		//If valid destination found
		IF(_MPD.CV[CvIndex].DepositFuncNumber <> E_FunctionNumber.F_BEGIN_FUNCTION) THEN
			_MPD.CV[CvIndex].HighestPriority := TRUE;
			_MPD.CV[CvIndex].State := E_MPD_CvStates.E_CV_OCCUPIED;
			IF(_DebugPrint) THEN _M_DebugPrint(0,'Recover->E_CV_OCCUPIED'); END_IF
			_M_GetPickupDepositFunctions := TRUE;
		END_IF
	ELSE	    
		//Normal functionality, get prioritized data  	
		_MPD.CV[CvIndex].PickupFuncNumber 	:= rPrioFunctions.PickupFunctionNumber;
		_MPD.CV[CvIndex].DepositFuncNumber 	:= rPrioFunctions.DepositFunctionNumber;
		_MPD.CV[CvIndex].HighestPriority 	:= rPrioFunctions.HighestPriority;
		_M_GetPickupDepositFunctions := TRUE;
	END_IF
ELSE
	_MPD.CV[CvIndex].PickupFuncNumber 	:= E_FunctionNumber.F_BEGIN_FUNCTION; 
	_MPD.CV[CvIndex].DepositFuncNumber 	:= E_FunctionNumber.F_BEGIN_FUNCTION;
	_MPD.CV[CvIndex].HighestPriority 	:= FALSE;
END_IF
END_METHOD

METHOD PRIVATE _M_IsErrorActive : BOOL

_M_IsErrorActive :=ElementData.ErrorData.FunctionErrorPending OR ElementData.ErrorData.ErrorState = E_ErrorState.ERROR;
END_METHOD

//check if Pickup or Deposit function is in error during takover or handover or if element is stoped
METHOD PRIVATE _M_IsErrorActiveOnPD : BOOL
VAR_INPUT
END_VAR
VAR
	i:INT;
	myElementNumber		: E_ElementNumber;
	myFunctionNumbers	: ARRAY [1..4] OF E_FunctionNumber;
END_VAR

//only check if an transport is activated
IF(_MPD.CV[GVL_MPD.CV_A].State = E_MPD_CvStates.E_CV_PICKUP) THEN
	myFunctionNumbers[1] := _MPD.CV[GVL_MPD.CV_A].PickupFuncNumber;
END_IF
IF(_MPD.CV[GVL_MPD.CV_A].State = E_MPD_CvStates.E_CV_DEPOSIT) THEN
	myFunctionNumbers[2] := _MPD.CV[GVL_MPD.CV_A].DepositFuncNumber;	
END_IF
IF(_MPD.CV[GVL_MPD.CV_B].State = E_MPD_CvStates.E_CV_PICKUP) THEN
	myFunctionNumbers[3] := _MPD.CV[GVL_MPD.CV_B].PickupFuncNumber;
END_IF
IF(_MPD.CV[GVL_MPD.CV_B].State = E_MPD_CvStates.E_CV_DEPOSIT) THEN
	myFunctionNumbers[4] := _MPD.CV[GVL_MPD.CV_B].DepositFuncNumber;
END_IF

(**************************************************************************************************************
//check that the deposit element, function or zone is in error	
**************************************************************************************************************)
FOR i:=1 TO 4 DO	
	IF(__ISVALIDREF(FunctionRegistry[myFunctionNumbers[i]].rSettingsFunction)) THEN
		myElementNumber := FunctionRegistry[myFunctionNumbers[i]].rSettingsFunction.eElementLink;
		IF(__ISVALIDREF(ElementRegistry[myElementNumber].rElementData))THEN
			IF(	ElementRegistry[myElementNumber].rElementData.ErrorData.FunctionErrorPending OR
				ElementRegistry[myElementNumber].rElementData.ErrorData.ErrorState = E_ErrorState.ERROR OR
				ElementRegistry[myElementNumber].rElementData.OperationState.eState = E_PositionState.STOPPED) THEN
				_M_IsErrorActiveOnPD := TRUE; //an error occured during and active TU transport (handover or takeover)
				EXIT; // no need to loock further
			END_IF		
		END_IF		
	END_IF
END_FOR
END_METHOD

METHOD PRIVATE _M_MPD_CvStates : BOOL
VAR_INPUT
	CvIndex 	: INT;  // 1=A, 2=B
END_VAR

CASE _MPD.CV[CvIndex].State OF
	
	E_MPD_CvStates.E_CV_INIT:		
		_MPD.CV[CvIndex].PickupFuncNumber := _MPD.CV[CvIndex].DepositFuncNumber := E_FunctionNumber.F_BEGIN_FUNCTION;
		_MPD.CV[CvIndex].HighestPriority := FALSE;		
		_MPD.CV[CvIndex].State := E_MPD_CvStates.E_CV_IDLE;
		IF(_DebugPrint) THEN _M_DebugPrint(CvIndex,'Idle');END_IF
		
	
	// idle, cv waiting for job assignment.
	E_MPD_CvStates.E_CV_IDLE:		
		
		IF _EntryReqActive OR _EntryModeActive OR ElementData.OperationState.eMode <> E_PositionMode.AUTO_MODE OR ElementData.OperationState.eState <> E_PositionState.STARTED THEN
			;//Do Nothing
		ELSIF (_MPD.CV[CvIndex].PickupFuncNumber <> E_FunctionNumber.F_BEGIN_FUNCTION AND _MPD.CV[CvIndex].DepositFuncNumber <> E_FunctionNumber.F_BEGIN_FUNCTION) THEN
				_MPD.CV[CvIndex].State := E_MPD_CvStates.E_CV_JOBASSIGNED;		
		ELSE
			//Get prioritized pickup and deposit function
			_M_GetPickupDepositFunctions(CvIndex, FALSE);			
		END_IF
		
		
	//Shuttle Conveyor has a job assigned, wait for shuttle to get into correct position
	E_MPD_CvStates.E_CV_JOBASSIGNED:
		//check that pickup position still is valid
		IF(NOT  _M_GetPickupDepositFunctions(CvIndex,TRUE(*Verify*))) THEN
			_MPD.CV[CvIndex].State := E_MPD_CvStates.E_CV_INIT;
		ELSIF( _MPD.CV[CvIndex].PosPickupReached) THEN			
			//ElementRegistry[E_ElementNumber.E_11_002_0206_00_0].rElement.fbDebugMsg.M_SendInfoMsg(CONCAT(CONCAT('Shuttle: ', GVL_MPD.CV_IxNAME[CvIndex]),CONCAT('. Pickup adjacent function: ', F_GetFunctionName(_SC.CV[CvIndex].PickupFuncNumber,0))));			
			_MPD.CV[CvIndex].State := E_MPD_CvStates.E_CV_PICKUP;			
		END_IF
	
	//Wait for pickup to be complete. ie transfer TU from pickup function on to the shuttle conveyor
	E_MPD_CvStates.E_CV_PICKUP:
		//Set links for  pickup adjacent function, to point towards correct Shuttle conveyor (CV A or CV B)
		_M_SetLinks(CvIndex,TRUE,FALSE,FALSE,ElementData.ErrorData.ErrorDataSet[7]);		
		IF(NOT CtrlIn.HoldPosition AND _M_CheckTransportComplete(_MPD.CV[CvIndex].State, CvIndex)) THEN 
			_MPD.CV[CvIndex].State := E_MPD_CvStates.E_CV_OCCUPIED;
			IF(_DebugPrint) THEN _M_DebugPrint(CvIndex,'->E_CV_OCCUPIED');END_IF
		END_IF
	
	// pickup complete, and shuttle conveyor occupied, wait for deposit function is reached
	E_MPD_CvStates.E_CV_OCCUPIED:
		//incase of recovery from abnormal shutdown or Semi Auto Mode
		IF(NOT _MPD.RequestMove OR _MPD.State = E_MPD_States.E_SEMI_MODE) THEN
			;//Wait 
		ELSIF( _MPD.CV[CvIndex].PosDepositReached) THEN
			//restore Pickup adjacent function to default
			_M_SetLinks(CvIndex,TRUE,FALSE,TRUE,ElementData.ErrorData.ErrorDataSet[7]);		
			IF(_DebugPrint) THEN _M_DebugPrint(CvIndex,CONCAT('->E_CV_DEPOSIT to function: ', F_GetFunctionName(_MPD.CV[CvIndex].DepositFuncNumber,0))); END_IF				
			_MPD.CV[CvIndex].State := E_MPD_CvStates.E_CV_DEPOSIT;
		END_IF
	
	E_MPD_CvStates.E_CV_DEPOSIT:	
		//incase of recovery from abnormal shutdown or Semi Auto Mode
		IF(NOT _MPD.RequestMove OR _MPD.State = E_MPD_States.E_SEMI_MODE) THEN
			_MPD.CV[CvIndex].State := E_MPD_CvStates.E_CV_OCCUPIED;
			IF(_DebugPrint) THEN _M_DebugPrint(CvIndex,'->E_CV_OCCUPIED'); END_IF
		END_IF
		//Set links for the deposit adjacent function, to point towards correct Shuttle conveyor (CV A or CV B)
		_M_SetLinks(CvIndex,FALSE,TRUE,FALSE,ElementData.ErrorData.ErrorDataSet[7]);		
		IF(NOT CtrlIn.HoldPosition AND _M_CheckTransportComplete(_MPD.CV[CvIndex].State, CvIndex)) THEN
			//restore deposit adjacent function to default
			_M_SetLinks(CvIndex,FALSE,TRUE,TRUE,ElementData.ErrorData.ErrorDataSet[7]);
			IF(_DebugPrint) THEN _M_DebugPrint(CvIndex,'->E_CV_DONE'); END_IF
			_MPD.CV[CvIndex].State := E_MPD_CvStates.E_CV_DONE;
		END_IF
	
	E_MPD_CvStates.E_CV_DONE:		
		IF(_MPD.State = E_MPD_States.E_CYCLE_COMPLETE) THEN						
			_MPD.CV[CvIndex].State := E_MPD_CvStates.E_CV_INIT;
		END_IF
	
	ELSE
		F_SetError( ErrorType:= E_ErrorType.ERROR, 	ErrorParam:= '_M_ShuttleCvStates sequence error' , ErrorMsg:= E_ErrorConv.SOFTWARE_ERROR, ErrorData:= ElementData.ErrorData.ErrorDataSet[7]);
	
END_CASE
END_METHOD

METHOD PRIVATE _M_MPD_Init : BOOL
VAR
	EmptyShuttleConv 	: ST_MPD_CV;
	i,j 				: INT;
	InitSuccess 		: BOOL :=TRUE;
END_VAR

VAR_INST
	InitDelay : TON; // Startup delay for the function(s) connected to the element to initialize 
END_VAR
// Init function, performed once at init
_MPD.CV[GVL_MPD.CV_A] := EmptyShuttleConv;
_MPD.CV[GVL_MPD.CV_B] := EmptyShuttleConv;
_MPD.State := 0;

//_SC.ShuttleFuncNumber					:= ElementData ConfigFunction.eFunctionNumber;
_MPD.CV[GVL_MPD.CV_A].CvFuncNumber	:= ElementData.MemberList.FunctionList[1].eFunctionNumber;
_MPD.CV[GVL_MPD.CV_B].CvFuncNumber	:= ElementData.MemberList.FunctionList[2].eFunctionNumber;

_MPD.CV[GVL_MPD.CV_A].Enabled		:= _MPD.CV[GVL_MPD.CV_A].CvFuncNumber <> E_FunctionNumber.F_BEGIN_FUNCTION;
_MPD.CV[GVL_MPD.CV_B].Enabled		:= _MPD.CV[GVL_MPD.CV_B].CvFuncNumber <> E_FunctionNumber.F_BEGIN_FUNCTION;
// Check if there is a Pick Desposit
IF(MPD_Config.MPD_Type = E_MotionPD_Type.E_Unknown) THEN
	F_SetError(ErrorType:= E_ErrorType.ERROR, 
				ErrorParam:= 'Motion PD type not defined', 
				ErrorMsg:= E_ErrorConv.CONFIGURATION_ERROR, 
				ErrorData:= ElementData.ErrorData.ErrorDataSet[NUMBER_OF_ERROR_SETS]); 
	InitSuccess:=FALSE;
END_IF
// -Check correct assignment in. Element has at least has a shuttle function + minimum one additional function
InitDelay(IN:=TRUE,PT:=T#10S);
IF(_MPD.CV[GVL_MPD.CV_A].CvFuncNumber = E_FunctionNumber.F_BEGIN_FUNCTION AND _MPD.CV[GVL_MPD.CV_B].CvFuncNumber = E_FunctionNumber.F_BEGIN_FUNCTION) THEN
	IF(InitDelay.Q) THEN
		F_SetError(ErrorType:= E_ErrorType.ERROR, 
					ErrorParam:= 'Element has not assigned CvA to an function', 
					ErrorMsg:= E_ErrorConv.CONFIGURATION_ERROR, 
					ErrorData:= ElementData.ErrorData.ErrorDataSet[NUMBER_OF_ERROR_SETS]); 
		InitDelay(IN:=FALSE);
	END_IF
	InitSuccess:=FALSE;
	RETURN;
END_IF
// Check configuration
// -Check that not the same function is assigned more than once
FOR i := 1 TO GVL_MPD.MAXPDs - 1 BY 1 DO 
	FOR j := i + 1 TO GVL_MPD.MAXPDs BY 1 DO
		IF (MPD_Config.ConvCFG[i].eFunctionNumber = MPD_Config.ConvCFG[j].eFunctionNumber  AND MPD_Config.ConvCFG[i].eFunctionNumber<>E_FunctionNumber.F_BEGIN_FUNCTION) THEN
			F_SetError(ErrorType:= E_ErrorType.ERROR, 
				ErrorParam:= CONCAT('Doublets configured in Config.ConvCFG index: ', INT_TO_STRING(i)) , 
				ErrorMsg:= E_ErrorConv.CONFIGURATION_ERROR, 
				ErrorData:= ElementData.ErrorData.ErrorDataSet[NUMBER_OF_ERROR_SETS]); 
				InitSuccess := FALSE;
		END_IF
	END_FOR
END_FOR
// Check configuration
// -check at least one of the EnableConv parameters are set
FOR i := 1 TO GVL_MPD.MAXPDs - 1 BY 1 DO	
	IF (MPD_Config.ConvCFG[i].eFunctionNumber <> E_FunctionNumber.F_BEGIN_FUNCTION AND
		(MPD_Config.ConvCFG[i].EnableConv[1]=FALSE AND  MPD_Config.ConvCFG[i].EnableConv[2]=FALSE)) THEN
			F_SetError(ErrorType:= E_ErrorType.ERROR, 
				ErrorParam:= CONCAT('Both EnableConv[x] in Config.ConvCFG index: ', INT_TO_STRING(i)) , 
				ErrorMsg:= E_ErrorConv.CONFIGURATION_ERROR, 
				ErrorData:= ElementData.ErrorData.ErrorDataSet[NUMBER_OF_ERROR_SETS]); 
				InitSuccess := FALSE;
	END_IF	
END_FOR	
// Check configuration
// -check that position is set within the valid range
FOR i := 1 TO GVL_MPD.MAXPDs - 1 BY 1 DO 
	FOR j:=GVL_MPD.CV_A TO GVL_MPD.CV_B DO
		IF (MPD_Config.ConvCFG[i].eFunctionNumber <> E_FunctionNumber.F_BEGIN_FUNCTION AND
			(MPD_Config.ConvCFG[i].EnableConv[j] AND (MPD_Config.ConvCFG[i].PositionConv < MPD_Config.DriveCFG.MinimumPosition OR MPD_Config.ConvCFG[i].PositionConv>MPD_Config.DriveCFG.MaximumPosition))) THEN
				F_SetError(ErrorType:= E_ErrorType.ERROR, 
					ErrorParam:= CONCAT('PositionConv in Config.ConvCFG index: ', INT_TO_STRING(i)), 
					ErrorMsg:= E_ErrorConv.CONFIGURATION_ERROR, 
					ErrorData:= ElementData.ErrorData.ErrorDataSet[NUMBER_OF_ERROR_SETS]); 
					InitSuccess := FALSE;
		END_IF
	END_FOR	
END_FOR
// Check the for invalid homing function should not be F_BegainFunction or set an error
IF MPD_Config.EncoderHoming.HomingFunctionNumber = E_FunctionNumber.F_BEGIN_FUNCTION AND MPD_Config.EncoderHoming.HomingEnable THEN
	F_SetError(ErrorType:= E_ErrorType.ERROR, 
					ErrorParam:= 'Invalid Homing Function number', 
					ErrorMsg:= E_ErrorConv.CONFIGURATION_ERROR, 
					ErrorData:= ElementData.ErrorData.ErrorDataSet[NUMBER_OF_ERROR_SETS]); 
					InitSuccess := FALSE;
END_IF	
// Check configuration
// Check pickup position offset
FOR i := 1 TO GVL_MPD.MAXPDs - 1 BY 1 DO 
	FOR j:=GVL_MPD.CV_A TO GVL_MPD.CV_B DO
		IF (MPD_Config.ConvCFG[i].eFunctionNumber <> E_FunctionNumber.F_BEGIN_FUNCTION AND MPD_Config.ConvCFG[i].EnableConv[j]) THEN
			
			IF(MPD_Config.MPD_Type = E_MotionPD_Type.E_ShuttleCar) THEN
				//PickupPositionOffset must be zero for shuttle cars
				IF(MPD_Config.MPD_Type = E_MotionPD_Type.E_ShuttleCar AND MPD_Config.ConvCFG[i].PickupPositionOffset<>0) THEN
					 F_SetError(ErrorType:= E_ErrorType.ERROR, 
						ErrorParam:= CONCAT('PickupPositionOffset<>0 . Config.ConvCFG index: ', INT_TO_STRING(i)), 
						ErrorMsg:= E_ErrorConv.CONFIGURATION_ERROR, 
						ErrorData:= ElementData.ErrorData.ErrorDataSet[NUMBER_OF_ERROR_SETS]); 
						InitSuccess := FALSE;
				END_IF
				//DepsitPositionOffset must be zero for shuttle cars
				 IF(MPD_Config.MPD_Type = E_MotionPD_Type.E_ShuttleCar AND MPD_Config.ConvCFG[i].DepsitPositionOffset<>0) THEN
					 F_SetError(ErrorType:= E_ErrorType.ERROR, 
						ErrorParam:= CONCAT('DepsitPositionOffset<>0 . Config.ConvCFG index: ', INT_TO_STRING(i)), 
						ErrorMsg:= E_ErrorConv.CONFIGURATION_ERROR, 
						ErrorData:= ElementData.ErrorData.ErrorDataSet[NUMBER_OF_ERROR_SETS]); 
						InitSuccess := FALSE;
				END_IF
			END_IF
			
			IF(MPD_Config.MPD_Type = E_MotionPD_Type.E_VerticalCv) THEN
				//PickupPositionOffset must be sane. ie between -200 and + 200
				IF(MPD_Config.ConvCFG[i].PickupPositionOffset > 200 AND MPD_Config.ConvCFG[i].PickupPositionOffset <-200) THEN
					F_SetError(ErrorType:= E_ErrorType.ERROR, 
						ErrorParam:= CONCAT('PickupPositionOffset +-200 in Config.ConvCFG index: ', INT_TO_STRING(i)), 
						ErrorMsg:= E_ErrorConv.CONFIGURATION_ERROR, 
						ErrorData:= ElementData.ErrorData.ErrorDataSet[NUMBER_OF_ERROR_SETS]); 
						InitSuccess := FALSE;
				END_IF
			END_IF
		END_IF
	END_FOR	
END_FOR
// Check CVCC, must be 0 for VC type
IF(MPD_Config.MPD_Type = E_MotionPD_Type.E_VerticalCv AND MPD_Config.CvCC <> 0) THEN
	F_SetError(ErrorType:= E_ErrorType.ERROR, 
				ErrorParam:= 'MPD_Config.CvCC must be set to 0', 
				ErrorMsg:= E_ErrorConv.CONFIGURATION_ERROR, 
				ErrorData:= ElementData.ErrorData.ErrorDataSet[NUMBER_OF_ERROR_SETS]); 
	InitSuccess:=FALSE;
END_IF

_M_MPD_Init := InitSuccess;
END_METHOD

METHOD PROTECTED _M_MPD_Mover : BOOL
VAR_INPUT
END_VAR
VAR
	i					: INT;
	DesiredPos			: DINT;	
	MoviDriveManual		: ST_MoviDriveManual;
END_VAR

VAR_INST
	CVInPosTimeout		: TON;//if position is not correct stop, set an error	
	ScMoveTimeout		: TON := (PT:=T#30S);	//Shuttle Car Move Timeout
	EntryReqState		: INT;
END_VAR

CASE EntryReqState OF
	0:	//Trig an entry request..
		IF(CtrlIn.RequestEntry) THEN 
			_EntryReqActive :=TRUE;
			EntryReqState := EntryReqState+1;
		END_IF
	1: // wait for position is reached
		IF(_MPD.EntryPosReached) THEN
			_EntryModeActive :=TRUE;
			_EntryReqActive :=FALSE;
			EntryReqState := EntryReqState+1;
		END_IF
	2: // Entry pos is reched, wait for operator to turn off key
		IF(NOT CtrlIn.RequestEntry) THEN
			_EntryModeActive :=FALSE;
			EntryReqState := EntryReqState+1;
		END_IF
	ELSE
		EntryReqState := 0;	
END_CASE


// Call Shuttle car mover...
// Manual Control
IF(_MPD.State = E_MPD_States.E_SEMI_MODE AND CtrlIn.SemiDriveCtrl.SemiManualMode) THEN 
	//Semi manual control
	MoviDriveManual.DriveFwd := CtrlIn.SemiDriveCtrl.SemiControlFWD;
	MoviDriveManual.DriveRev := CtrlIn.SemiDriveCtrl.SemiControlREV;
	MoviDriveManual.EmergencyDrive := FALSE;
ELSE
	//Normal Manual control
	MoviDriveManual.DriveFwd := HW_Inputs.ManualControl.DriveFwd;
	MoviDriveManual.DriveRev := HW_Inputs.ManualControl.DriveRev;
	MoviDriveManual.EmergencyDrive := HW_Inputs.ManualControl.EmergencyDrive;
END_IF



IF( NOT ProBoxSystem.EMULATION_ENABLED) THEN	
		
	//Request to move Normal operation
	IF _MPD.RequestMove AND NOT _EntryModeActive THEN 
		fbMPDMover.M_MoveAbsolute(
			mPosition		:= _MPD.RequestPosValue, 
			mVelocity		:= MPD_Config.DriveCFG.DriveParameter[_MPD.DriveParameterIndex].Velocity, 
			mAcceleration	:= MPD_Config.DriveCFG.DriveParameter[_MPD.DriveParameterIndex].Acceleration, 
			mDeceleration	:= MPD_Config.DriveCFG.DriveParameter[_MPD.DriveParameterIndex].Deceleration, 
			mJerk			:= MPD_Config.DriveCFG.DriveParameter[_MPD.DriveParameterIndex].Jerk,
			ErrorData 		:= ElementData.ErrorData.ErrorDataSet[5]);
	
	//Request move to entry
	ELSIF _EntryReqActive AND NOT _MPD.RequestMove AND _MPD.State = E_MPD_States.E_IDLE THEN 
		fbMPDMover.M_MoveAbsolute(
			mPosition		:= CtrlIn.RequestEntryPos, //EntryPosition, 
			mVelocity		:= MPD_Config.DriveCFG.DriveParameter[_MPD.DriveParameterIndex].Velocity, 
			mAcceleration	:= MPD_Config.DriveCFG.DriveParameter[_MPD.DriveParameterIndex].Acceleration, 
			mDeceleration	:= MPD_Config.DriveCFG.DriveParameter[_MPD.DriveParameterIndex].Deceleration, 
			mJerk			:= MPD_Config.DriveCFG.DriveParameter[_MPD.DriveParameterIndex].Jerk,
			ErrorData 		:= ElementData.ErrorData.ErrorDataSet[5]);
	END_IF
	
	fbMPDMover(
		ErrorPending			:= _M_IsErrorActive(), 
		ElementOperationState	:= ElementData.OperationState,
		DisableEnableDrive 		:= (NOT _MPD.RequestMove AND NOT _EntryReqActive) OR _M_IsErrorActiveOnPD(), 
		DriveCFG				:= MPD_Config.DriveCFG,
		ManualControl			:= MoviDriveManual,		  
		DriveInputs				:= HW_Inputs.DriveInputs,		
		EmgStopAxisTrig 		:= EmergencyStop,
		Done 					=> _MPD.Locked, 
		Aborted 				=> _MPD.MotionAborted,
		ErrorData 				:= ElementData.ErrorData.ErrorDataSet[5]);
	
	
	
	_MPD.ActualPosValue := LREAL_TO_DINT( fbMPDMover.ActPos);
END_IF	
	

//-----------------------------------------------------------------------------
// Set interface variables used in ShuttleState and ShuttleCVStates
//-----------------------------------------------------------------------------
FOR i:=GVL_MPD.CV_A TO GVL_MPD.CV_B DO
			
	//Pickup position reached?
	DesiredPos := M_GetDesiredPosition(_MPD.CV[i].PickupFuncNumber, i, TRUE,FALSE);
	_MPD.CV[i].PosPickupReached := M_CheckDesiredPosition(DesiredPos) AND _MPD.Locked AND _MPD.RequestMove AND _MPD.CV[i].PickupFuncNumber > E_FunctionNumber.F_BEGIN_FUNCTION;
	
	//Deposit position reached?
	DesiredPos := M_GetDesiredPosition(_MPD.CV[i].DepositFuncNumber, i, FALSE, TRUE);	
	_MPD.CV[i].PosDepositReached := M_CheckDesiredPosition(DesiredPos) AND _MPD.Locked AND _MPD.RequestMove AND _MPD.CV[i].DepositFuncNumber > E_FunctionNumber.F_BEGIN_FUNCTION;
END_FOR

	//Idle Position reached?
	_MPD.IdlePosReached := M_CheckDesiredPosition(MPD_Config.IdlePosition) AND _MPD.Locked AND MPD_Config.EnableIdlePosition;

	//Entry Position reached?
	_MPD.EntryPosReached := M_CheckDesiredPosition(CtrlIn.RequestEntryPos) AND _MPD.Locked;

//-----------------------------------------------------------------------------	
// Error handling: Check car movement is performed within acceptable time 
//-----------------------------------------------------------------------------	
	
//Check shuttle Car movement Timeout
ScMoveTimeout(IN:=_MPD.RequestMove AND NOT _MPD.Locked AND (ElementData.OperationState.eState = E_PositionState.STARTED OR ElementData.OperationState.eState = E_PositionState.STOPPING), 
				PT:= MPD_Config.TimeOutMove);
IF(ScMoveTimeout.Q) THEN
	F_SetError( ErrorType:= E_ErrorType.ERROR, 	ErrorParam:= 'Movement Timeout' , (* Could not get to the destination with in expected time*) 
				ErrorMsg:= E_ErrorConv.TIMEOUT, ErrorData:= ElementData.ErrorData.ErrorDataSet[4]);
	ScMoveTimeout(IN:=FALSE);
END_IF


//-----------------------------------------------------------------------------	
// Error handling: Timeout during takeover or handover. Note: the Shuttle car servo shall stop immediately
// If element is not in error and not adjacent function, then it is somthiing else that makes the transport not possible to finalize (could be that the deposit function is disabled..)
//-----------------------------------------------------------------------------
CVInPosTimeout(	IN:= NOT _M_IsErrorActive() AND NOT _M_IsErrorActiveOnPD() AND _MPD.RequestMove AND ( _MPD.State = E_MPD_States.E_PICKINGUP OR _MPD.State = E_MPD_States.E_DEPOSITING),
				PT:= MPD_Config.TimeOutMove); 
IF(CVInPosTimeout.Q) THEN		 
	F_SetError(E_ErrorType.ERROR,'Timeout during Pickup or deposit',E_ErrorConv.TIMEOUT,ElementData.ErrorData.ErrorDataSet[4]);
END_IF 

	
//-----------------------------------------------------------------------------
//Emulation shuttle car posioning
//-----------------------------------------------------------------------------
END_METHOD

METHOD PRIVATE _M_MPD_States : BOOL
VAR_INPUT
END_VAR


VAR	
	i		: INT;
	OtherCv	: ARRAY[1..2] OF INT := [GVL_MPD.CV_B,GVL_MPD.CV_A];	
END_VAR

VAR_INST
	EnterIdlePosTmr		: TON := (PT:= T#2S); //delay before entering Idle position	
END_VAR
EnterIdlePosTmr();


CASE _MPD.State OF
	
	//---------------------------------------------------------------------------------------------------
	E_MPD_States.E_INIT:
		_MPD.RequestMove := FALSE;
		_MPD.State:=E_MPD_States.E_IDLE;
		
	
		
	//---------------------------------------------------------------------------------------------------
	// Waiting for job to do	
	E_MPD_States.E_IDLE: 
		EnterIdlePosTmr.IN:=FALSE;
		_M_AutoAdjustVCHeight(FALSE,FALSE,TRUE (*Reset*), FALSE);
				
		//Check if we can proceed...
		IF(ElementData.OperationState.eState <> E_PositionState.STARTED OR ElementData.OperationState.eMode <> E_PositionMode.AUTO_MODE OR
		   _EntryReqActive OR _EntryModeActive)  THEN
			//do nothing, but wait
 			_MPD.RequestMove	:= FALSE;	
		
		//Semi automatic or semi manual mode
		ELSIF(CtrlIn.SemiDriveCtrl.SemiAutoMode OR CtrlIn.SemiDriveCtrl.SemiManualMode) THEN			
			_MPD.State := E_MPD_States.E_SEMI_MODE;			
			IF(_DebugPrint) THEN _M_DebugPrint(0,CONCAT('->E_SEMI_MODE : ', TO_STRING(_MPD.RequestPosValue))); END_IF
	
		//Normal operation, picking up
		ELSIF( _MPD.CV[GVL_MPD.CV_A].State = E_MPD_CvStates.E_CV_PICKUP OR _MPD.CV[GVL_MPD.CV_B].State = E_MPD_CvStates.E_CV_PICKUP) THEN 
			_MPD.State := E_MPD_States.E_PICKINGUP;
			
		//Normal operation, Depositing
		ELSIF( _MPD.CV[GVL_MPD.CV_A].State = E_MPD_CvStates.E_CV_DEPOSIT OR _MPD.CV[GVL_MPD.CV_B].State = E_MPD_CvStates.E_CV_DEPOSIT) THEN 
			_MPD.State := E_MPD_States.E_DEPOSITING;
			
		//Normal operation, check if an job is assigned to CV A or CV B
		ELSIF( _MPD.CV[GVL_MPD.CV_A].State = E_MPD_CvStates.E_CV_JOBASSIGNED OR _MPD.CV[GVL_MPD.CV_B].State = E_MPD_CvStates.E_CV_JOBASSIGNED) THEN		
			// Element has no error pending and wheres a job to do	
			_MPD.State := E_MPD_States.E_START_PICKUP;						
		
		//check if CV A or CV B is occupied
		ELSIF( _MPD.CV[GVL_MPD.CV_A].State = E_MPD_CvStates.E_CV_OCCUPIED OR _MPD.CV[GVL_MPD.CV_B].State = E_MPD_CvStates.E_CV_OCCUPIED) THEN	 
			_MPD.State := E_MPD_States.E_START_DEPOSIT;		
			
		//If no active jobs move to idle position	
		ELSIF (MPD_Config.EnableIdlePosition) THEN
			EnterIdlePosTmr.IN := NOT _MPD.IdlePosReached AND NOT _EntryReqActive AND NOT _M_IsErrorActive();
			IF(EnterIdlePosTmr.Q) THEN			
					// Set desired Shuttle car position
					_MPD.RequestPosValue := MPD_Config.IdlePosition;
					// Release shuttle car brake
					_MPD.RequestMove := TRUE;
			ELSE
				_MPD.RequestMove := FALSE;
			END_IF
		END_IF
	
	
	
		//---------------------------------------------------------------------------------------------------
		// Semi automatic mode	
		E_MPD_States.E_SEMI_MODE:
			IF ((NOT CtrlIn.SemiDriveCtrl.SemiAutoMode AND NOT CtrlIn.SemiDriveCtrl.SemiManualMode)OR
				(ElementData.OperationState.eMode <> E_PositionMode.AUTO_MODE)) THEN
				_MPD.RequestMove := FALSE;
				_MPD.State := E_MPD_States.E_IDLE;
				IF(_DebugPrint) THEN _M_DebugPrint(0,CONCAT('->E_IDLE : ', TO_STRING(_MPD.RequestPosValue))); END_IF		
			END_IF		
		
		
		
		
	//---------------------------------------------------------------------------------------------------
	// Decide prioirty for A and B	
	E_MPD_States.E_START_PICKUP:
				
		FOR i:=GVL_MPD.CV_A TO GVL_MPD.CV_B DO			
			IF( _M_IsErrorActive()=FALSE ) THEN  //element has no error pending
				IF(_MPD.CV[i].State = E_MPD_CvStates.E_CV_JOBASSIGNED AND (_MPD.CV[i].HighestPriority  OR _MPD.CV[OtherCv[i]].State = E_MPD_CvStates.E_CV_OCCUPIED))THEN
					// Set desired Shuttle car position
					_MPD.RequestPosValue := M_GetDesiredPosition(_MPD.CV[i].PickupFuncNumber, i, TRUE,FALSE);
					// Release shuttle car brake
					_MPD.RequestMove := TRUE;
					//move to next state
					_MPD.State := E_MPD_States.E_MOVE_TO_PICKUP;					
					IF(_DebugPrint) THEN _M_DebugPrint(0,CONCAT('->E_MOVE_TO_PICKUP : ', TO_STRING(_MPD.RequestPosValue))); END_IF
					EXIT;					
				END_IF	
			END_IF				
		END_FOR
		

	
	//---------------------------------------------------------------------------------------------------	
	E_MPD_States.E_MOVE_TO_PICKUP:
		
		IF(_MPD.CV[GVL_MPD.CV_A].State <> E_MPD_CvStates.E_CV_JOBASSIGNED AND _MPD.CV[GVL_MPD.CV_B].State <> E_MPD_CvStates.E_CV_JOBASSIGNED) THEN
			_MPD.State:=E_MPD_States.E_IDLE; //start over, Shuttle CV states may not be fulfiled anymore.  
		ELSE			
			//Check if shuttle car is in position
			FOR i:=GVL_MPD.CV_A TO GVL_MPD.CV_B DO
				IF(_MPD.CV[i].PosPickupReached ) THEN				
					//position reached				
					_MPD.State := E_MPD_States.E_PICKUP_POSITION_REACHED;				
					IF(_DebugPrint) THEN _M_DebugPrint(0,'->E_PICKUP_POSITION_REACHED'); END_IF	
					EXIT;			
				END_IF								
			END_FOR
		END_IF
			
		
		
	//---------------------------------------------------------------------------------------------------	
	E_MPD_States.E_PICKUP_POSITION_REACHED:
		//At this point only check that MPD locked the position, as the acutal position may change if AutoAdjustVCHeight is used.
		IF(_MPD.Locked AND NOT _MPD.MotionAborted) THEN
			_MPD.State := E_MPD_States.E_PICKINGUP;
		END_IF

	//---------------------------------------------------------------------------------------------------		
	E_MPD_States.E_PICKINGUP:
	
		//Adjust VC height
		_MPD.RequestPosValue := _MPD.RequestPosValue + _M_AutoAdjustVCHeight(TRUE,FALSE,FALSE,FALSE);
		//wait for pickup is complete
		//there can be a situation where we have a parallell transport of CvA and CvB, so wait till conveyors finishing transport
		IF (_MPD.CV[GVL_MPD.CV_A].State <> E_MPD_CvStates.E_CV_PICKUP AND _MPD.CV[GVL_MPD.CV_B].State <> E_MPD_CvStates.E_CV_PICKUP) THEN						
			_MPD.State:=E_MPD_States.E_IDLE; //start over, and see the other shuttle CV (CV_A or CV_B) should be picked up						
			IF(_DebugPrint) THEN _M_DebugPrint(0,'E_PICKINGUP->E_IDLE'); END_IF						
		END_IF
		
		//in case motion was aborted/interupted. it may be so that SC/VC position is changed, check position is maintained. 
		IF(_MPD.MotionAborted) THEN
			_MPD.State:=E_MPD_States.E_PICKUP_POSITION_REACHED;
			IF(_DebugPrint) THEN _M_DebugPrint(0,'E_PICKINGUP->E_PICKUP_POSITION_REACHED'); END_IF
		END_IF
		
	//---------------------------------------------------------------------------------------------------		
	E_MPD_States.E_START_DEPOSIT: 
			
		FOR i:=GVL_MPD.CV_A TO GVL_MPD.CV_B DO
			IF(_M_IsErrorActive()=FALSE AND _MPD.CV[i].State = E_MPD_CvStates.E_CV_OCCUPIED AND (_MPD.CV[i].HighestPriority OR _MPD.CV[OtherCv[i]].State = E_MPD_CvStates.E_CV_DONE))THEN				
				// reqest shuttle car position
				_MPD.RequestPosValue := M_GetDesiredPosition(_MPD.CV[i].DepositFuncNumber, i, FALSE,TRUE);
				// Release shuttle car brake
				_MPD.RequestMove := TRUE;
				_MPD.State := E_MPD_States.E_MOVE_TO_DEPOSIT;
				IF(_DebugPrint) THEN _M_DebugPrint(0,CONCAT('E_START_DEPOSIT->E_MOVE_TO_DEPOSIT : ',  TO_STRING(_MPD.RequestPosValue))); END_IF
				EXIT;
			END_IF				
		END_FOR
	
	
	//---------------------------------------------------------------------------------------------------
	//Check if shuttle car is in position for depositing		
	E_MPD_States.E_MOVE_TO_DEPOSIT:
		//Check if shuttle car is in position
		FOR i:=GVL_MPD.CV_A TO GVL_MPD.CV_B DO
			IF(_MPD.CV[i].PosDepositReached AND _MPD.CV[i].State = E_MPD_CvStates.E_CV_DEPOSIT) THEN //if deposit position is reached, and CV_A or CV_B has reacted				
				//position reached				
				_MPD.State := E_MPD_States.E_DEPOSIT_POSITION_REACHED;
				IF(_DebugPrint) THEN _M_DebugPrint(0,CONCAT('E_MOVE_TO_DEPOSIT->E_DEPOSIT_POSITION_REACHED: ', GVL_MPD.CV_IxNAME[i])); END_IF
				EXIT; //break for loop				
			END_IF			
		END_FOR
	
			
	//---------------------------------------------------------------------------------------------------		
	E_MPD_States.E_DEPOSIT_POSITION_REACHED:
	//At this point only check that MPD locked the position, as the acutal position may change if AutoAdjustVCHeight is used.
		IF(_MPD.Locked AND NOT _MPD.MotionAborted) THEN
			_MPD.State:=E_MPD_States.E_DEPOSITING;	
		END_IF
	
	//---------------------------------------------------------------------------------------------------	
	E_MPD_States.E_DEPOSITING:
		//incase of recovery from abnormal shutdown or Semi Auto Mode	
		IF(NOT _MPD.RequestMove) THEN
			_MPD.State := E_MPD_States.E_START_DEPOSIT;
		END_IF
	
		//Adjust VC height
		_MPD.RequestPosValue := _MPD.RequestPosValue + _M_AutoAdjustVCHeight(FALSE,TRUE,FALSE,FALSE);
		
		//wait for depositing is complete		
		FOR i:=GVL_MPD.CV_A TO GVL_MPD.CV_B DO
			IF ((_MPD.CV[i].State = E_MPD_CvStates.E_CV_PICKUP OR _MPD.CV[OtherCv[i]].State = E_MPD_CvStates.E_CV_PICKUP) OR 
				(_MPD.CV[i].State = E_MPD_CvStates.E_CV_DEPOSIT OR _MPD.CV[OtherCv[i]].State = E_MPD_CvStates.E_CV_DEPOSIT))THEN
				// in the case we do an pickup in parallell with deposit (shuttle with 2 conveyors)
				;// do nothing but wait.							
			ElSIF (_MPD.CV[i].State = E_MPD_CvStates.E_CV_DONE AND _MPD.CV[OtherCv[i]].State = E_MPD_CvStates.E_CV_OCCUPIED) THEN
				// Go back and set the next deposit position for the shuttle car
				_MPD.State:=E_MPD_States.E_START_DEPOSIT;  	
				IF(_DebugPrint) THEN _M_DebugPrint(0,'E_DEPOSITING->E_START_DEPOSIT'); END_IF 	
			ELSIF( (_MPD.CV[i].State = E_MPD_CvStates.E_CV_DONE AND _MPD.CV[otherCv[i]].State <= E_MPD_CvStates.E_CV_IDLE) OR
				   (_MPD.CV[i].State = E_MPD_CvStates.E_CV_DONE AND _MPD.CV[otherCv[i]].State = E_MPD_CvStates.E_CV_DONE)) THEN	
					//proceed to next step			
					_MPD.State:=E_MPD_States.E_CYCLE_COMPLETE;
					IF(_DebugPrint) THEN _M_DebugPrint(0,'E_DEPOSITING->E_CYCLE_COMPLETE'); END_IF
			END_IF
		END_FOR
		
		//in case motion was aborted/interupted. it may be so that SC/VC position is changed, check position is maintained. 
		IF(_MPD.MotionAborted) THEN
			_MPD.State:=E_MPD_States.E_DEPOSIT_POSITION_REACHED;
		END_IF
		
		
	//---------------------------------------------------------------------------------------------------
	E_MPD_States.E_CYCLE_COMPLETE:
				
		_MPD.State:=E_MPD_States.E_INIT;
		
	ELSE
		F_SetError( ErrorType:= E_ErrorType.ERROR, 	ErrorParam:= '_M_ShuttleStates sequence error' , ErrorMsg:= E_ErrorConv.SOFTWARE_ERROR, ErrorData:= ElementData.ErrorData.ErrorDataSet[7]);
	
END_CASE
END_METHOD

METHOD PROTECTED _M_SemiDriveControl : BOOL
VAR_INPUT
END_VAR

IF(_MPD.State <> E_MPD_States.E_SEMI_MODE) THEN
	MemSet(ADR(fbMPDMover.SemiDriveControl),0, SIZEOF(fbMPDMover.SemiDriveControl));
ELSE
	fbMPDMover.SemiDriveControl.SemiAutoMode			:= CtrlIn.SemiDriveCtrl.SemiAutoMode AND NOT CtrlIn.SemiDriveCtrl.SemiManualMode;
	fbMPDMover.SemiDriveControl.SemiManualMode 			:= CtrlIn.SemiDriveCtrl.SemiManualMode AND NOT CtrlIn.SemiDriveCtrl.SemiAutoMode;
	fbMPDMover.SemiDriveControl.SemiTrigMoveAbs		 	:= CtrlIn.SemiDriveCtrl.SemiAutoEnableDrive;
	fbMPDMover.SemiDriveControl.SemiAutoHalt 			:= CtrlIn.SemiDriveCtrl.SemiAutoHalt;	
	//set request move
	IF(fbMPDMover.SemiDriveControl.SemiAutoMode) THEN
		//Semi auto mode
		_MPD.RequestMove := CtrlIn.SemiDriveCtrl.SemiAutoEnableDrive;
		_MPD.RequestPosValue := CtrlIn.SemiDriveCtrl.SemiAutoPositionToGo;					
	ELSE
		//Semi Man mode
		_MPD.RequestMove := FALSE;
	END_IF
	
	//Reset input variables in case user did'nt...
	CtrlIn.SemiDriveCtrl.SemiAutoHalt 					:= FALSE;
	IF(fbMPDMover.PositioningState = E_PositioningState.POSITIONING_ABSOLUTE) THEN	
		CtrlIn.SemiDriveCtrl.SemiAutoEnableDrive			:= FALSE;	
	END_IF
END_IF
END_METHOD

// Replace the deposit or pickup position adjacent functionnumber to point toward CVA or CVB
METHOD PRIVATE _M_SetAdjacentFunction : BOOL
VAR_INPUT
	ScCvFunction		: E_FunctionNumber; //the shuttle car conveyor function
	AdjacentFunction	: E_FunctionNumber; //the pickup or deposit function to change
	SearchFunctions		: ARRAY[1..3] OF E_FunctionNumber;
	RestoreToDefault	: BOOL;
END_VAR

VAR
	rFuncSettings  	: REFERENCE TO ST_CFG_Function;		//the pickup or deposit function where to replace the adjacent side
	rConfigSettings	: REFERENCE TO ST_CFG_Function;
	i:INT;
END_VAR

//

rFuncSettings REF= FunctionRegistry[AdjacentFunction].rSettingsFunction;
rConfigSettings REF= FunctionRegistry[AdjacentFunction].rFunction.ConfigFunction; 

//Replace the adjacent side of the deposit function to point towards the Shuttle conveyor A
IF(__ISVALIDREF(rFuncSettings) AND __ISVALIDREF(rConfigSettings)) THEN
	IF(NOT RestoreToDefault) THEN
		FOR i:= 1 TO 4 DO
			IF(	rFuncSettings.eAdjacentFunctionNumberSide[i] <> E_FunctionNumber.F_BEGIN_FUNCTION AND
				(rFuncSettings.eAdjacentFunctionNumberSide[i] = SearchFunctions[1] OR
				 rFuncSettings.eAdjacentFunctionNumberSide[i] = SearchFunctions[2] OR
				 rFuncSettings.eAdjacentFunctionNumberSide[i] = SearchFunctions[3] )) THEN
				 
					rFuncSettings.eAdjacentFunctionNumberSide[i] := ScCvFunction;
					_M_SetAdjacentFunction :=TRUE;
					//EXIT;
			END_IF			
		END_FOR
	// restore to default
	ELSE 
		rFuncSettings.eAdjacentFunctionNumberSide := rConfigSettings.eAdjacentFunctionNumberSide;				
	END_IF	
	
END_IF
END_METHOD

// Setup links, adjacent sides on shuttle car towards the pickup and deposition funciton
METHOD PRIVATE _M_SetLinks : BOOL
VAR_INPUT
	//CvAFuncNumb		: E_FunctionNumber;
	SC_CV_Index 		: INT; // 1 = A, 2 = B  
	SetPickupLinks		: BOOL; 
	SetDepositLinks		: BOOL; 
	RestorToDefault		: BOOL;
END_VAR
VAR_IN_OUT
	ErrorData 				: ST_ErrorDataSet; // Error data
END_VAR
VAR
	ReplaceFunctions	: ARRAY[1..3] OF E_FunctionNumber;	
END_VAR
	ReplaceFunctions[1] := _MPD.CV[GVL_MPD.CV_A].CvFuncNumber;	//the Shuttle Car Conveyor A functionNumber
	ReplaceFunctions[2] := _MPD.CV[GVL_MPD.CV_B].CvFuncNumber;	//the Shuttle Car Conveyor B functionNumber
	ReplaceFunctions[3] := E_FunctionNumber.F_BEGIN_FUNCTION;	//Spare, to remove?
	
	
	//Sanity check
	IF( NOT __ISVALIDREF(FunctionRegistry[_MPD.CV[SC_CV_Index].CvFuncNumber].rSettingsFunction)) THEN
		F_SetError(	ErrorType := E_ErrorType.ERROR,	ErrorParam := 'Setup Pickup transport link',ErrorMsg := E_ErrorConv.INCORRECT_POSITION, ErrorData := ErrorData);
		_M_SetLinks:= FALSE;
		RETURN;
	END_IF
		
	IF(NOT RestorToDefault AND SetPickupLinks) THEN		
		//Setup SettingsFunctions parameters for shuttle car conveyor		
		FunctionRegistry[_MPD.CV[SC_CV_Index].CvFuncNumber].rSettingsFunction.ePrevFunctionNumber := _MPD.CV[SC_CV_Index].PickupFuncNumber;
		FunctionRegistry[_MPD.CV[SC_CV_Index].CvFuncNumber].rSettingsFunction.eNextFunctionNumber := E_FunctionNumber.F_BEGIN_FUNCTION;
		
		//Set adjacent sides on shuttle conveyor	
		IF( M_GetConveyorDirection(_MPD.CV[SC_CV_Index].PickupFuncNumber) = E_PickupDepositSide.LeftSide) THEN
			//Pickup on left side -> drive Forward 
			FunctionRegistry[_MPD.CV[SC_CV_Index].CvFuncNumber].rSettingsFunction.eAdjacentFunctionNumberSide[1] := _MPD.CV[SC_CV_Index].PickupFuncNumber;
			FunctionRegistry[_MPD.CV[SC_CV_Index].CvFuncNumber].rSettingsFunction.eAdjacentFunctionNumberSide[2] := E_FunctionNumber.F_BEGIN_FUNCTION;	
		ELSE                 
			//Pickup on right side -> drive Reverse
			FunctionRegistry[_MPD.CV[SC_CV_Index].CvFuncNumber].rSettingsFunction.eAdjacentFunctionNumberSide[1] := E_FunctionNumber.F_BEGIN_FUNCTION;
			FunctionRegistry[_MPD.CV[SC_CV_Index].CvFuncNumber].rSettingsFunction.eAdjacentFunctionNumberSide[2] := _MPD.CV[SC_CV_Index].PickupFuncNumber;					
		END_IF		
	END_IF
	
	IF(NOT RestorToDefault AND SetDepositLinks) THEN
		//Setup SettingsFunctions parameters for shuttle car conveyor
		FunctionRegistry[_MPD.CV[SC_CV_Index].CvFuncNumber].rSettingsFunction.ePrevFunctionNumber := E_FunctionNumber.F_BEGIN_FUNCTION;		
		FunctionRegistry[_MPD.CV[SC_CV_Index].CvFuncNumber].rSettingsFunction.eNextFunctionNumber := _MPD.CV[SC_CV_Index].DepositFuncNumber;
		//Set adjacent sides on shuttle conveyor
		IF( M_GetConveyorDirection(_MPD.CV[SC_CV_Index].DepositFuncNumber) = E_PickupDepositSide.RightSide) THEN
			//Deposit on left side -> drive Forward		
			FunctionRegistry[_MPD.CV[SC_CV_Index].CvFuncNumber].rSettingsFunction.eAdjacentFunctionNumberSide[1] := E_FunctionNumber.F_BEGIN_FUNCTION;
			FunctionRegistry[_MPD.CV[SC_CV_Index].CvFuncNumber].rSettingsFunction.eAdjacentFunctionNumberSide[2] := _MPD.CV[SC_CV_Index].DepositFuncNumber;	
		ELSE
			//Deposit on Right side -> drive reverse                 
			FunctionRegistry[_MPD.CV[SC_CV_Index].CvFuncNumber].rSettingsFunction.eAdjacentFunctionNumberSide[1] := _MPD.CV[SC_CV_Index].DepositFuncNumber;
			FunctionRegistry[_MPD.CV[SC_CV_Index].CvFuncNumber].rSettingsFunction.eAdjacentFunctionNumberSide[2] := E_FunctionNumber.F_BEGIN_FUNCTION;					
		END_IF		
	END_IF
	 
	
	
	// change the adjacent function number for the pickup function, to point to the correct shuttle conveyor A or B
	IF(NOT RestorToDefault AND SetPickupLinks) THEN
		IF( NOT _M_SetAdjacentFunction(_MPD.CV[SC_CV_Index].CvFuncNumber,_MPD.CV[SC_CV_Index].PickupFuncNumber,ReplaceFunctions,FALSE) OR
			NOT _M_SetTransportlink(_MPD.CV[SC_CV_Index].PickupFuncNumber,_MPD.CV[SC_CV_Index].CvFuncNumber,0,FALSE,FALSE)) THEN				
				F_SetError(	ErrorType := E_ErrorType.ERROR,	ErrorParam := 'Setup Pickup transport link',ErrorMsg := E_ErrorConv.INCORRECT_POSITION, ErrorData := ErrorData);
				_M_SetLinks:= FALSE;		
				RETURN;
		END_IF
	END_IF

	// change the adjacent function number for the deposit function	
	IF(NOT RestorToDefault AND SetDepositLinks) THEN		
		IF( NOT _M_SetAdjacentFunction(_MPD.CV[SC_CV_Index].CvFuncNumber,_MPD.CV[SC_CV_Index].DepositFuncNumber,ReplaceFunctions, FALSE)OR 
			NOT _M_SetTransportlink(_MPD.CV[SC_CV_Index].DepositFuncNumber,0,_MPD.CV[SC_CV_Index].CvFuncNumber,FALSE,FALSE)) THEN
				F_SetError(	ErrorType := E_ErrorType.ERROR,	ErrorParam := 'Setup Deposit transport link',ErrorMsg := E_ErrorConv.INCORRECT_POSITION, ErrorData := ErrorData);
				_M_SetLinks:= FALSE;
				RETURN;
		END_IF
	END_IF
	
	//----------------------------------------------------------------------------------------------------------------------------
	//restore to default
	IF(RestorToDefault AND SetPickupLinks ) THEN
		_M_SetAdjacentFunction(0,_MPD.CV[SC_CV_Index].PickupFuncNumber,ReplaceFunctions, TRUE);
		_M_SetTransportlink(_MPD.CV[SC_CV_Index].PickupFuncNumber,0,0,FALSE,TRUE);
		//and for the shuttle conveyor it self
		_M_SetTransportlink(_MPD.CV[SC_CV_Index].CvFuncNumber,0,0,TRUE,FALSE);		
	END_IF
	IF(RestorToDefault AND SetDepositLinks) THEN
		_M_SetAdjacentFunction(0,_MPD.CV[SC_CV_Index].DepositFuncNumber,ReplaceFunctions, TRUE);
		_M_SetTransportlink(_MPD.CV[SC_CV_Index].DepositFuncNumber,0,0,TRUE,FALSE);
		//and for the shuttle conveyor it self
		_M_SetTransportlink(_MPD.CV[SC_CV_Index].CvFuncNumber,0,0,TRUE,TRUE);
	END_IF

	
	_M_SetLinks:= TRUE;  //method run successfully, without any error
END_METHOD

//Set function interface, Previous and Next function, for adjacent functions to point to wards the Shuttle conveyor
//This is needed when shuttle car is configured with two shuttle conveyors (A and B)
METHOD PRIVATE _M_SetTransportlink : BOOL
VAR_INPUT	
	AdjacentFunction	: E_FunctionNumber; //the pickup or deposit function to change
	NextFunction		: E_FunctionNumber;
	PreviusFunction		: E_FunctionNumber;
	RevertPrevious		: BOOL; // restore to default
	RevertNext			: BOOL; // restore to default
END_VAR

VAR
	rFuncSettings	: REFERENCE TO ST_CFG_Function;
	rConfigSettings	: REFERENCE TO ST_CFG_Function;
	rFunctInterface : REFERENCE TO ST_FunctionInterface;
END_VAR

//

rFuncSettings REF= FunctionRegistry[AdjacentFunction].rSettingsFunction; 
rConfigSettings REF= FunctionRegistry[AdjacentFunction].rFunction.ConfigFunction;
rFunctInterface REF= FunctionRegistry[AdjacentFunction].rFunctionInterface; 

IF( NOT __ISVALIDREF(rFuncSettings) OR NOT __ISVALIDREF(rFunctInterface) OR NOT __ISVALIDREF(rConfigSettings)) THEN
	RETURN;
ELSE
	_M_SetTransportlink :=TRUE;
END_IF


//Replace the adjacent side of the deposit function to point towards the Shuttle conveyor A

	
IF(NOT RevertPrevious AND NOT RevertNext) THEN
			
	IF(NextFunction <> E_FunctionNumber.F_BEGIN_FUNCTION) THEN
		//IF(rFuncSettings.eNextFunctionNumber <> E_FunctionNumber.F_BEGIN_FUNCTION) THEN
		rFuncSettings.eNextFunctionNumber := NextFunction;
		rFunctInterface.In.eNextFunctionNumber := NextFunction;			
	END_IF
	
	IF(PreviusFunction <> E_FunctionNumber.F_BEGIN_FUNCTION) THEN
		rFuncSettings.ePrevFunctionNumber := PreviusFunction;			
		rFunctInterface.In.ePrevFunctionNumber := PreviusFunction;			
	END_IF
	
ELSE
	//restore to default
	IF(RevertPrevious) THEN
		rFuncSettings.ePrevFunctionNumber := rConfigSettings.ePrevFunctionNumber;
		rFunctInterface.In.ePrevFunctionNumber := E_FunctionNumber.F_BEGIN_FUNCTION;
	END_IF			
	IF(RevertNext) THEN
		rFuncSettings.eNextFunctionNumber := rConfigSettings.eNextFunctionNumber;
		rFunctInterface.In.eNextFunctionNumber := E_FunctionNumber.F_BEGIN_FUNCTION;
	END_IF		
END_IF
END_METHOD

ACTION A_Init:
(**************************************************************************************
 * 	NAME		A_Init
 * 	FUNCTION	Initialize function
 **************************************************************************************)
 

// Init ongoing - Wait until init is released (Sequencial startup)
IF NOT ElementData.Init AND ElementData.InitRunning THEN	
	_MPDlInitDone:=FALSE;	
END_IF		

IF(ElementData.Init AND NOT _MPDlInitDone) THEN
	// Init shuttle mover
	fbMPDMover.M_Init();
	_MPDlInitDone := _M_MPD_Init();
END_IF
END_ACTION

ACTION A_OutputMapping:
(**************************************************************************************
 * 	NAME		A_OutputMapping
 * 	FUNCTION	Output mapping
 **************************************************************************************)
 
(**************************************************************************************
   Hardware outputs
***************************************************************************************)
HW_Outputs.MotionOutputLow			:= fbMPDMover.AxisMotionOutputLow;
HW_Outputs.MotionOutputHigh			:= fbMPDMover.AxisMotionOutputHigh;
HW_Outputs.DriveOutputs				:= fbMPDMover.DriveOutputs;
HW_Outputs.EnableDrive				:= fbMPDMover.EnableDrive;

CtrlOut.EntryRequestProcessed		:= _EntryModeActive;
CtrlOut.MotionRunning 				:= fbMPDMover.Busy AND NOT fbMPDMover.Done; 
CtrlOut.MotionComplete				:= fbMPDMover.Done;

(**************************************************************************************
   Order outputs (Commands to corresponding element)
***************************************************************************************)
// init FunctionInterface
MEMSET(ADR(FunctionInterface.Out.FunctionOrders),0,SIZEOF(ST_FunctionOrders)); 

//Manual mode
IF(ElementData.OperationState.eMode = E_PositionMode.MANUAL_MODE) THEN
	FunctionInterface.Out.FunctionOrders.Enable			:= HW_Inputs.ManualControl.Conv[GVL_MPD.CV_A].ConvFwd OR HW_Inputs.ManualControl.Conv[GVL_MPD.CV_A].ConvRev;
	FunctionInterface.Out.FunctionOrders.ReqDriveRun 	:= HW_Inputs.ManualControl.Conv[GVL_MPD.CV_A].ConvFwd OR HW_Inputs.ManualControl.Conv[GVL_MPD.CV_A].ConvRev;
	FunctionInterface.Out.FunctionOrders.ReqDriveDirection := HW_Inputs.ManualControl.Conv[GVL_MPD.CV_A].ConvFwd AND NOT HW_Inputs.ManualControl.Conv[GVL_MPD.CV_A].ConvRev;	// TRUE = FWD
	FunctionInterface.Out.FunctionOrders.ReqSpeed 		:= 100; // normal speed E_ProBoxMotorSpeed.NORMAL
	
	FunctionInterface.Out.FunctionOrders.Enable_34		:= HW_Inputs.ManualControl.Conv[GVL_MPD.CV_B].ConvFwd OR HW_Inputs.ManualControl.Conv[GVL_MPD.CV_B].ConvRev;
	FunctionInterface.Out.FunctionOrders.ReqDriveRun_34	:= HW_Inputs.ManualControl.Conv[GVL_MPD.CV_B].ConvFwd OR HW_Inputs.ManualControl.Conv[GVL_MPD.CV_B].ConvRev;
	FunctionInterface.Out.FunctionOrders.ReqDriveDirection_34 := HW_Inputs.ManualControl.Conv[GVL_MPD.CV_B].ConvFwd AND NOT HW_Inputs.ManualControl.Conv[GVL_MPD.CV_B].ConvRev;	// TRUE = FWD
	FunctionInterface.Out.FunctionOrders.ReqSpeed_34 	:= 100; // normal speed E_ProBoxMotorSpeed.NORMAL
END_IF


//Auto mode
IF(ElementData.OperationState.eMode = E_PositionMode.AUTO_MODE AND (ElementData.OperationState.eState = E_PositionState.STARTED OR ElementData.OperationState.eState = E_PositionState.STOPPING)) THEN
	// Axis 1-2 (shuttle car CV A) drive run
	FunctionInterface.Out.FunctionOrders.Enable := NOT _M_IsErrorActive() AND 
													( M_CheckDesiredPosition(M_GetDesiredPosition(_MPD.CV[GVL_MPD.CV_A].PickupFuncNumber, GVL_MPD.CV_A,TRUE,FALSE)) OR M_CheckDesiredPosition(M_GetDesiredPosition(_MPD.CV[GVL_MPD.CV_A].DepositFuncNumber, GVL_MPD.CV_A, FALSE, TRUE))) AND
													(_MPD.State=E_MPD_States.E_DEPOSITING OR _MPD.State = E_MPD_States.E_PICKINGUP) AND
													(_MPD.CV[GVL_MPD.CV_A].State = E_MPD_CvStates.E_CV_PICKUP OR _MPD.CV[GVL_MPD.CV_A].State = E_MPD_CvStates.E_CV_DEPOSIT);
	FunctionInterface.Out.FunctionOrders.ReqDriveRun := FALSE;
	FunctionInterface.Out.FunctionOrders.ReqDriveDirection := FALSE;
	FunctionInterface.Out.FunctionOrders.ReqSpeed := 0;
	
	// Axis 3-4 (shuttle car CV B) drive run
	FunctionInterface.Out.FunctionOrders.Enable_34 := NOT _M_IsErrorActive() AND
													( M_CheckDesiredPosition(M_GetDesiredPosition(_MPD.CV[GVL_MPD.CV_B].PickupFuncNumber, GVL_MPD.CV_B,TRUE,FALSE)) OR M_CheckDesiredPosition(M_GetDesiredPosition(_MPD.CV[GVL_MPD.CV_B].DepositFuncNumber, GVL_MPD.CV_B,FALSE,TRUE))) AND 
													(_MPD.State=E_MPD_States.E_DEPOSITING OR _MPD.State = E_MPD_States.E_PICKINGUP) AND
													(_MPD.CV[GVL_MPD.CV_B].State = E_MPD_CvStates.E_CV_PICKUP OR _MPD.CV[GVL_MPD.CV_B].State = E_MPD_CvStates.E_CV_DEPOSIT);
	FunctionInterface.Out.FunctionOrders.ReqDriveRun_34 := FALSE;
	FunctionInterface.Out.FunctionOrders.ReqDriveDirection_34 := FALSE;
	FunctionInterface.Out.FunctionOrders.ReqSpeed_34 := 0;	
END_IF



(**************************************************************************************
   AddOn outputs
***************************************************************************************)
// This function provide no AddOn functionality
;
END_ACTION

//Check if the actual position is at the desired position including allowed variations (EncoderHysterisis)
METHOD PUBLIC M_CheckDesiredPosition : BOOL
VAR_INPUT
	DesiredPos			: DINT; //the desired shuttle position to check if is within hysterisis boundaries
END_VAR
VAR
	MaxVal,MinVal,AdjVal : DINT;
END_VAR

MaxVal := DesiredPos + (MPD_Config.EncoderHysterisis);
MinVal := DesiredPos - (MPD_Config.EncoderHysterisis);

AdjVal := _M_AutoAdjustVCHeight(FALSE,FALSE,FALSE,TRUE);
IF(AdjVal<0) THEN
	MinVal:= MinVal + AdjVal;
ELSE
	MaxVal:= MaxVal + AdjVal;
END_IF


M_CheckDesiredPosition := 	(DesiredPos > 0 AND DesiredPos <16#7FFFFFFF) (*maximum possible value*) AND
							(_MPD.ActualPosValue <= MaxVal) AND 
							(_MPD.ActualPosValue >= MinVal);
END_METHOD

METHOD PUBLIC M_GetConveyorDirection : E_PickupDepositSide
VAR_INPUT	
	FunctionNumber			: E_FunctionNumber;
END_VAR
VAR
	i:INT;
END_VAR
M_GetConveyorDirection:= E_PickupDepositSide.Unknown;

IF(FunctionNumber = E_FunctionNumber.F_BEGIN_FUNCTION) THEN RETURN; END_IF

FOR i:=1 TO GVL_MPD.MAXPDs DO
	IF(MPD_Config.ConvCFG[i].eFunctionNumber = FunctionNumber ) THEN
		M_GetConveyorDirection:= MPD_Config.ConvCFG[i].Side;
		EXIT;
	END_IF		
END_FOR
END_METHOD

//Get the absolute encoder position value for the shuttle car set in configuration
METHOD PUBLIC M_GetDesiredPosition : DINT
VAR_INPUT	
	FunctionNumber		: E_FunctionNumber;
	CvIndex				: INT; // 1=A, 2=B
	PickUp				: BOOL;	//Is VC picking up, if so then also consider the PickupPositionOffset value
	Depsit				: BOOL; //Is VC Depositing, if so then aslo consideer the DepostPositionOffset value;
END_VAR
VAR_OUTPUT
	Valid				: BOOL; //The retured position/distance is valid 
END_VAR
VAR
	i:INT;
END_VAR

M_GetDesiredPosition:= 16#7FFFFFFF;
Valid:=FALSE;
IF(FunctionNumber = E_FunctionNumber.F_BEGIN_FUNCTION) THEN RETURN; END_IF

FOR i:=1 TO GVL_MPD.MAXPDs DO
	IF(MPD_Config.ConvCFG[i].eFunctionNumber = FunctionNumber ) THEN
		Valid:=TRUE;
		M_GetDesiredPosition:= MPD_Config.ConvCFG[i].PositionConv;
		IF(CvIndex = GVL_MPD.CV_B AND MPD_Config.MPD_Type = E_MotionPD_Type.E_ShuttleCar) THEN
			M_GetDesiredPosition := M_GetDesiredPosition - MPD_Config.CvCC;
		END_IF
		
		IF(MPD_Config.MPD_Type = E_MotionPD_Type.E_VerticalCv) THEN
			IF(PickUp)THEN
				M_GetDesiredPosition := M_GetDesiredPosition + MPD_Config.ConvCFG[i].PickupPositionOffset;
			ELSIF(Depsit)THEN
				M_GetDesiredPosition := M_GetDesiredPosition + MPD_Config.ConvCFG[i].DepsitPositionOffset;
			END_IF
		END_IF
		
		EXIT;
		
	END_IF		
END_FOR
END_METHOD

PROPERTY PUBLIC P_AutoAdjustVcHeight : REFERENCE TO ST_AutoAdjustVcHeight
GET
P_AutoAdjustVcHeight REF= _AutoAdjustVcHeight;
END_GET
SET
_AutoAdjustVcHeight := P_AutoAdjustVcHeight;
END_SET
END_PROPERTY

//Get property of _MPD data container
PROPERTY PUBLIC P_GetMpdData : REFERENCE TO ST_MPD
GET
P_GetMpdData REF= _MPD;
END_GET
END_PROPERTY

//Set/Get the driveParameter index to select the motion profile of ST_CFG_MPD_Drive.DriveParameter[x]
//Make sure that an prifile is configed properly befor applying a new DriveParameterIndex
PROPERTY PUBLIC P_SetDriveParameterIndex : UINT
GET
P_SetDriveParameterIndex := _MPD.DriveParameterIndex;
END_GET
SET
IF(P_SetDriveParameterIndex>0)THEN
	_MPD.DriveParameterIndex := P_SetDriveParameterIndex;
END_IF
END_SET
END_PROPERTY

END_FUNCTION_BLOCK

// ---- 20_Product/20_ProBox/22_ProMove/03_Controls/12_MotionPickAndDeposit/FB_MPD_PriorityControl.TcPOU
//Get the 2 most prioritized pickup functions
FUNCTION_BLOCK FB_MPD_PriorityControl
VAR_INPUT
	ConfigPDs				: REFERENCE TO ARRAY[1..GVL_MPD.MAXPDs] OF ST_CFG_PDs;		
	CvAFunctionNumber		: E_FunctionNumber;	 //the shuttel Conveyor A function number
	CvBFunctionNumber		: E_FunctionNumber;	 //the shuttel Conveyor B function number
	OverrideFunctions 		: ARRAY[1..GVL_MPD.MAXPDs] OF BOOL;	//Pickup functions that is set with higher prioirty
	IgnoreDepositCheck		: ARRAY[1..GVL_MPD.MAXPDs] OF BOOL; //Deposit functions that is set to not check conditions.
	MPD_Type				: E_MotionPD_Type;		// Motion PD type
END_VAR
VAR_OUTPUT
	
	CV_A					: ST_PrioFunctions;
	CV_B					: ST_PrioFunctions;
		
END_VAR
VAR
	_fbFifo			:FB_MergingFiFo;	
	
END_VAR
VAR_TEMP
	i:INT;
	InternalDisables: BOOL;//ARRAY [1..GVL_MPD.MAXCONV] OF BOOL;
	DisabledFunctions: ARRAY [1..GVL_MPD.MAXPDs] OF BOOL;
	AdjacentFunctionNumbers	: ARRAY [1..GVL_MPD.MAXPDs] OF E_FunctionNumber;	// The function numbers of all adjacent functions
	DepositFunction : E_FunctionNumber;
	
	PickupFunctionNumberA	: E_FunctionNumber;	//the function number that has the highest pickup priority
	PickupFunctionNumberB	: E_FunctionNumber;	//the function number that has the second highest pickup priority
	DepositFunctionNumberA	: E_FunctionNumber;
	DepositFunctionNumberB	: E_FunctionNumber;
	
	CvA_Enabled				: BOOL; //is conveyor A enabled (zone, function, element)	
	CvB_Enabled				: BOOL; //is conveyor B enabled (zone, function, element)
	
	CV_PickupEnabled		: ARRAY[1..2] OF BOOL;
	CV_DepositEnabled		: ARRAY[1..2] OF BOOL;
	CV_A_IsAssigned			: BOOL;
	MPD_ConfigIx			: INT; //index of the deposit function in MPD Config struct
	_IgnoreDepositCheck		: BOOL;
END_VAR

	
	//extract deposit/pickup functions
	FOR i:=1 TO GVL_MPD.MAXPDs BY 1 DO
		AdjacentFunctionNumbers[i] := ConfigPDs[i].eFunctionNumber;		 
	END_FOR	
 		
	//convert from override to disable	
	_M_ConvertOverrideToDisables(OverrideFunctions:=OverrideFunctions, DisabledFunctions=>DisabledFunctions);
	
	CV_A.PickupFunctionNumber:=CV_A.DepositFunctionNumber:=E_FunctionNumber.F_BEGIN_FUNCTION;	
	CV_B.PickupFunctionNumber:=CV_B.DepositFunctionNumber:=E_FunctionNumber.F_BEGIN_FUNCTION;
	CV_A.HighestPriority:=CV_B.HighestPriority:=FALSE;
	
	MEMSET(ADR(InternalDisables),0,SIZEOF(InternalDisables));
	// Get Prioirty of the pickup function that has the higest priority
	FOR i:=1 TO GVL_MPD.MAXPDs BY 1 DO			
		DepositFunction  := M_GetDepositFunction(AdjacentFunctionNumbers[i],0,FALSE,MPD_ConfigIndex=>MPD_ConfigIx);
		_IgnoreDepositCheck := SEL(MPD_ConfigIx>0 AND MPD_ConfigIx<=GVL_MPD.MAXPDs,FALSE,IgnoreDepositCheck[MPD_ConfigIx]); 
		InternalDisables := _M_IsEnabled(AdjacentFunctionNumbers[i])= FALSE;
		InternalDisables := InternalDisables OR (_M_IsEnabled(DepositFunction)= FALSE);		
		InternalDisables := InternalDisables OR _M_CheckConditions(AdjacentFunctionNumbers[i], DepositFunction, _IgnoreDepositCheck);
		_fbFifo(FunctionNumber:=AdjacentFunctionNumbers[i],Disable:=DisabledFunctions[i] OR InternalDisables);
	END_FOR
	
	//Set outputs A	
	//Get the most prioritized pickup funciton number.
	PickupFunctionNumberA  := _fbFifo.ePrevFunctionNumber;
	DepositFunctionNumberA := M_GetDepositFunction(PickupFunctionNumberA,0,FALSE);
	
	//Set outputs B
	//Get the second most prioritized pickup function number.
	PickupFunctionNumberB  := _fbFifo.M_GetFifoIndex(2);
	DepositFunctionNumberB := M_GetDepositFunction(PickupFunctionNumberB,0,FALSE);
	
	
	CvA_Enabled := _M_IsEnabled(CvAFunctionNumber);
	CvB_Enabled := _M_IsEnabled(CvBFunctionNumber);
	
	
	//Check the most prioritized task can be set to conveyor X
	IF(PickupFunctionNumberA <> E_FunctionNumber.F_BEGIN_FUNCTION) THEN
		CV_PickupEnabled := _M_GetConveyorEnabled(ConfigPDs,PickupFunctionNumberA);
		CV_DepositEnabled := _M_GetConveyorEnabled(ConfigPDs,DepositFunctionNumberA);
		IF (CV_PickupEnabled[1] AND CV_DepositEnabled[1] AND CvA_Enabled) THEN // set the TU with most priority to CV A
			CV_A.PickupFunctionNumber := PickupFunctionNumberA;		
			CV_A.DepositFunctionNumber := DepositFunctionNumberA;
			CV_A.HighestPriority := TRUE;
			CV_A_IsAssigned:=TRUE;
		ELSIF (CV_PickupEnabled[2] AND CV_DepositEnabled[2] AND CvB_Enabled) THEN // set the TU with most priority to CV B
			CV_B.PickupFunctionNumber := PickupFunctionNumberA;
			CV_B.DepositFunctionNumber := DepositFunctionNumberA;
			CV_B.HighestPriority := TRUE;
		END_IF
	END_IF
	
	//Check the second most prioritized task can be set to conveyor X 
	IF(PickupFunctionNumberB <> E_FunctionNumber.F_BEGIN_FUNCTION) THEN
		CV_PickupEnabled := _M_GetConveyorEnabled(ConfigPDs,PickupFunctionNumberB);
		CV_DepositEnabled := _M_GetConveyorEnabled(ConfigPDs,DepositFunctionNumberB);	
		IF(CV_A_IsAssigned) THEN
			IF (CV_PickupEnabled[2] AND CV_DepositEnabled[2] AND CvB_Enabled) THEN // set the TU with 2nd most priority to CV B
				CV_B.PickupFunctionNumber := PickupFunctionNumberB;
				CV_B.DepositFunctionNumber := DepositFunctionNumberB;
				CV_B.HighestPriority := FALSE;
			END_IF
		ELSE
			IF (CV_PickupEnabled[1] AND CV_DepositEnabled[1] AND CvA_Enabled) THEN // set the TU with 2nd most priority to CV A
				CV_A.PickupFunctionNumber := PickupFunctionNumberB;
				CV_A.DepositFunctionNumber := DepositFunctionNumberB;
				CV_A.HighestPriority := FALSE;
			END_IF
		END_IF
	END_IF

//Check that the adjacent function is an valid pickup position,
//Check that the destination is free and not in error
//Return: TRUE if the function shuld be disabled
METHOD PRIVATE _M_CheckConditions : BOOL
VAR_INPUT
	PickupFunctionNumber	: E_FunctionNumber;	 //the adjacent function number	
	DepositFunction 		: E_FunctionNumber;	
	IgnoreDepositCheck		: BOOL; //TRUE = Deposit function is not validated and being considered as valid.		
END_VAR

VAR		
	PickupZoneIndex 	: INT;
	DepositZoneIndex 	: INT;	
	
	TuDestination 		: E_FunctionNumber;
	TmpZoneData 		: ST_ZoneData;
	TmpTranspState		: E_TransportState;
	//ConditionValid 		: BOOL;
	ConditionNotValid : BOOL;
	i:INT;
	TU_DataIndex :DINT;
	DepositElementNumber	: E_ElementNumber;
	
END_VAR
	
	// sanity checks
	IF( NOT __ISVALIDREF(FunctionRegistry[PickupFunctionNumber].rFunction) OR
		NOT __ISVALIDREF(FunctionRegistry[DepositFunction].rFunction) OR	   
	    PickupFunctionNumber = E_FunctionNumber.F_BEGIN_FUNCTION ) OR 
		DepositFunction=E_FunctionNumber.F_BEGIN_FUNCTION THEN 
			_M_CheckConditions:=TRUE;
			RETURN;
	 END_IF
	
	// ------------------------------------------------------------------------------------
	//Check if the deposit function is set as "ignore condition checks"
	IF(IgnoreDepositCheck) THEN
		_M_CheckConditions:=FALSE; //Stop conditional check and return as the deposit function is valid. 
		RETURN;
	END_IF
	
	// ------------------------------------------------------------------------------------	
	
	
	//get the deposit zone index closest to the shuttle
	F_PB_GetAdjacentFunctionZoneIndex(DepositFunction,CvAFunctionNumber,FALSE,TRUE,DepositZoneIndex);		
	IF(	DepositZoneIndex =0) THEN
		F_PB_GetAdjacentFunctionZoneIndex(DepositFunction,CvBFunctionNumber,FALSE,TRUE,DepositZoneIndex);		
	END_IF
		
	
	//Sanity check
	IF(DepositZoneIndex<=0 OR DepositZoneIndex >NUMBER_OF_ZONES_PER_FUNCTION) THEN		
		_M_CheckConditions := TRUE; //True=> Pickup position should be disabled 	
		RETURN;
	END_IF
	
	(**************************************************************************************************************		
	//check that the Deposit function is ready to takeover TU
	**************************************************************************************************************)
	TmpTranspState := F_PB_GetTransportControlDataRef(DepositFunction,DepositZoneIndex).eTransportState;
	IF( NOT (TmpTranspState = E_TransportState.IDLE OR TmpTranspState = E_TransportState.FREE OR TmpTranspState = E_TransportState.TAKEOVER)) THEN
 		ConditionNotValid := TRUE; //True=> Pickup position should be disabled because deposit function is not ready
	END_IF
	
	
	//TODO
	//check functionInterface.in.PreviusFunction?? risk for deadlock if condition is set in merging flow control??
	
	//TODO
	// check Pickup position for errors on Element
	
	(**************************************************************************************************************
	//Check that the deposit function all zones are not Busy
	**************************************************************************************************************)
	IF(__ISVALIDREF(FunctionRegistry[DepositFunction].rSettingsFunction)) THEN
		FOR i:=1 TO FunctionRegistry[DepositFunction].rSettingsFunction.NumberOfZones DO
	 		TmpZoneData := F_GetZoneData(DepositFunction, i);
			 IF(	TmpZoneData.TransportControlData.eHandOverState = E_HandOverState.ACTIVE OR
					TmpZoneData.TransportControlData.eHandOverState = E_HandOverState.INTERRUPTED OR
					TmpZoneData.TransportControlData.eHandOverState = E_HandOverState.STOP OR
					TmpZoneData.TransportControlData.eTakeOverState = E_TakeOverState.ACTIVE OR
					TmpZoneData.TransportControlData.eTakeOverState = E_TakeOverState.INTERRUPTED OR
					TmpZoneData.TransportControlData.eTakeOverState = E_TakeOverState.STOP) THEN
				ConditionNotValid := TRUE;	//True=> Pickup position should be disabled	because any zone is not ready		 
			 END_IF
		END_FOR
	ELSE
		ConditionNotValid := TRUE; //True=> Pickup position should be disabled
	END_IF
 
	(**************************************************************************************************************
	//check that the deposit function is not occupied	
	**************************************************************************************************************)	
	IF(__ISVALIDREF(FunctionRegistry[DepositFunction].Zone[DepositZoneIndex].refZoneData)) THEN
		IF( FunctionRegistry[DepositFunction].Zone[DepositZoneIndex].refZoneData.TransportControlData.Occupied) THEN
			ConditionNotValid := TRUE; //True=> Pickup position should be disabled because the deposit function is occupied
		END_IF	
	ELSE
		ConditionNotValid := TRUE; //True=> Pickup position should be disabled
	END_IF
	
	
	(**************************************************************************************************************
	//check that the deposit element, function or zone is in error	
	**************************************************************************************************************)
	IF(__ISVALIDREF(FunctionRegistry[DepositFunction].rSettingsFunction)) THEN
		DepositElementNumber := FunctionRegistry[DepositFunction].rSettingsFunction.eElementLink;
		IF(__ISVALIDREF(ElementRegistry[DepositElementNumber].rElementData))THEN
			IF(ElementRegistry[DepositElementNumber].rElementData.ErrorData.FunctionErrorPending OR ElementRegistry[DepositElementNumber].rElementData.ErrorData.ErrorState = E_ErrorState.ERROR) THEN
				ConditionNotValid := TRUE; //True=> Pickup position should be disabled because the deposit element or function or zone(s) is in error
			END_IF
		ELSE
			ConditionNotValid := TRUE; //True=> Pickup position should be disabled
		END_IF		
	END_IF
	
	
	
	(**************************************************************************************************************
	// Check that the deposit function has enabled transport and enabled takeover	
	**************************************************************************************************************)		
	IF ( NOT FunctionRegistry[DepositFunction].rFunction.ZoneInterface[DepositZoneIndex].In.Enable.Transport OR
		 NOT FunctionRegistry[DepositFunction].rFunction.ZoneInterface[DepositZoneIndex].In.Enable.TakeOver) THEN
			ConditionNotValid := TRUE; //True=> Pickup position should be disabled because deposit functin is not ready		
	END_IF
	
	
	(**************************************************************************************************************
	//check that the destinations function are not in error	???
	**************************************************************************************************************)
	(*ConditionValid := FALSE;
	FOR i:=1 TO E_FunctionNumber.F_BEGIN_EXTERN_FUNCTION DO
		IF(PossibleDestinations[i] <> E_FunctionNumber.F_BEGIN_FUNCTION) THEN		
			IF(__ISVALIDREF(FunctionRegistry[PossibleDestinations[i]].Zone[DepositZoneIndex].refZoneData) AND 
			   __ISVALIDREF(FunctionRegistry[PossibleDestinations[i]].rSettingsFunction) ) THEN
						
				FOR i:=1 TO FunctionRegistry[PossibleDestinations[i]].rSettingsFunction.NumberOfZones DO		
					ConditionValid := FunctionRegistry[DepositFunction].Zone[1].refZoneData.ErrorData.ErrorState = E_ErrorState.OPERATIONAL;
				END_FOR
			END_IF
		END_IF
	END_FOR
	ConditionNotValid := ConditionNotValid OR NOT ConditionValid;*)
	
	
	(**************************************************************************************************************
	//set output	
	**************************************************************************************************************)
	_M_CheckConditions := ConditionNotValid; //True=> Pickup position should be disabled
END_METHOD

METHOD PRIVATE _M_ConvertOverrideToDisables
VAR_IN_OUT	
	OverrideFunctions 		: ARRAY[1..GVL_MPD.MAXPDs] OF BOOL;
END_VAR
VAR_OUTPUT
	DisabledFunctions		: ARRAY[1..GVL_MPD.MAXPDs] OF BOOL;
END_VAR
VAR
	OverridesActive:BOOL;
	i:int;
END_VAR

	//convert from override to disable	
	FOR i:=1 TO GVL_MPD.MAXPDs DO
		IF(OverrideFunctions[i]) THEN
			OverridesActive:=TRUE;
		END_IF
	END_FOR
	
	IF(OverridesActive) THEN
		MEMSET(ADR(DisabledFunctions), BOOL_TO_BYTE(TRUE),SIZEOF(DisabledFunctions));	
		FOR i:=1 TO GVL_MPD.MAXPDs DO
			DisabledFunctions[i]:= NOT OverrideFunctions[i];
		END_FOR
	END_IF
END_METHOD

//check that the deposit / pickup position is enabled( for Convayor A or B can reach the position)
METHOD PRIVATE _M_GetConveyorEnabled : ARRAY[1..2] OF BOOL
VAR_INPUT
	ConfigPDs				: REFERENCE TO ARRAY[1..GVL_MPD.MAXPDs] OF ST_CFG_PDs;
	FunctionNumber			: E_FunctionNumber;
END_VAR
VAR
	i:INT;
END_VAR

IF(FunctionNumber = E_FunctionNumber.F_BEGIN_FUNCTION) THEN RETURN; END_IF

FOR i:=1 TO GVL_MPD.MAXPDs DO
	IF(ConfigPDs[i].eFunctionNumber = FunctionNumber ) THEN
		_M_GetConveyorEnabled[1]:= ConfigPDs[i].EnableConv[1];
		_M_GetConveyorEnabled[2]:= ConfigPDs[i].EnableConv[2];
		EXIT;
	END_IF		
END_FOR
END_METHOD

//Get enable status. Zone, Function or element disabled via SIS interface
METHOD PRIVATE _M_IsEnabled : BOOL
VAR_INPUT
	FuncNumber 		: E_FunctionNumber;
END_VAR

VAR
	myElementNumber : E_ElementNumber;
	
END_VAR

_M_IsEnabled := FALSE;

IF(FuncNumber = E_FunctionNumber.F_BEGIN_FUNCTION) THEN
	RETURN;
END_IF

IF( NOT __ISVALIDREF(FunctionRegistry[FuncNumber].rSettingsFunction)) THEN
	RETURN;
END_IF

myElementNumber := FunctionRegistry[FuncNumber].rSettingsFunction.eElementLink;


IF( NOT __ISVALIDREF(ElementRegistry[myElementNumber].rElementInterface) OR 
	NOT __ISVALIDREF(FunctionRegistry[FuncNumber].rFunctionInterface) OR
	NOT __ISVALIDREF(FunctionRegistry[FuncNumber].Zone[1].refZoneInterface)) THEN
	RETURN;
END_IF

_M_IsEnabled := ElementRegistry[myElementNumber].rElementInterface.In.ElementEnable AND 
				FunctionRegistry[FuncNumber].rFunctionInterface.In.FunctionEnable AND
				FunctionRegistry[FuncNumber].Zone[1].refZoneInterface.In.ZoneEnable;
END_METHOD

METHOD PUBLIC M_CheckConditions : BOOL
VAR_INPUT
	PickupFunctionNumber	: E_FunctionNumber;	 //the adjacent function number	
	DepositFunction 		: E_FunctionNumber;	
	IgnoreDepositCheck		: BOOL; //TRUE = Deposit function is not validated and being considered as valid.		
END_VAR
M_CheckConditions := _M_CheckConditions(PickupFunctionNumber,DepositFunction,IgnoreDepositCheck);
END_METHOD

//Get the corresponding Deposit Function based on the destination of the TU located on pickup function  
METHOD PUBLIC M_GetDepositFunction : E_FunctionNumber
VAR_INPUT	
	PickupFunctionNumber	: E_FunctionNumber;
	ZoneIndex				: INT;	// Set to 0 in order for the method to lookup the zone index
	RecoverUsingLastTUix	: BOOL; // in case of recover, we may need to use the LastTU_DataIndex
END_VAR
VAR_OUTPUT
	MPD_ConfigIndex			: INT; // the index of the MPD index
END_VAR

VAR		
	TuDestination	: E_FunctionNumber;
	ZoneIx:INT;
	TU_DataIndex:DINT;
	i:INT;
	j:INT;
END_VAR
MPD_ConfigIndex:=0;
// sanity checks
	IF(NOT __ISVALIDREF(FunctionRegistry[PickupFunctionNumber].rFunction) OR	   
	   PickupFunctionNumber = E_FunctionNumber.F_BEGIN_FUNCTION) THEN
		RETURN;
	 END_IF
	 	 
	 
	//Get the Zone index of the pickupFunction that is closest to the shuttle function 
	//This is also an implicit check that the pickupFunction has its "next function" or "previous function" set to shuttle function
	//Check both Shuttle convayor A and B as in F_ConfigPosition we dont know if the pickup position pointing towards CV A or CV B 	 
	IF(ZoneIndex=0) THEN
		F_PB_GetAdjacentFunctionZoneIndex(PickupFunctionNumber,CvAFunctionNumber,TRUE,FALSE,ZoneIx);
		//ZoneIx := FunctionRegistry[PickupFunctionNumber].rFunction.M_GetTransportData(meFunctionNumber := CvAFunctionNumber).ZoneNumber;
		IF(ZoneIx = 0) THEN
			F_PB_GetAdjacentFunctionZoneIndex(PickupFunctionNumber,CvBFunctionNumber,TRUE, FALSE,ZoneIx);
			//ZoneIx := FunctionRegistry[PickupFunctionNumber].rFunction.M_GetTransportData(meFunctionNumber := CvBFunctionNumber).ZoneNumber;
		END_IF			
		//sanity check
		IF(ZoneIx=0) THEN
			RETURN; //Not possible determine the zone, it may be because the pickup position not has its next position set towards the shuttle CV A or CV B
		END_IF
	ELSE
		ZoneIx := ZoneIndex;
	END_IF	
	
	//get the TU index of the pickup adjacentFunction
	TU_DataIndex := F_PB_GetTransportControlDataRef(PickupFunctionNumber,ZoneIx).TU_DataIndex; 
	IF(RecoverUsingLastTUix AND TU_DataIndex=0) THEN // try with last TU_DataIndex when recover
		TU_DataIndex := F_PB_GetTransportControlDataRef(PickupFunctionNumber,ZoneIx).LastTU_DataIndex;
	END_IF
	
	//Get the TU destination number from TU table
	TuDestination := TU_Table.TU_DataTable[TU_DataIndex].Destination[1].eFunctionNumber;
	
	//************************************************************************************************
	//Search for Deposit function
	//************************************************************************************************
	//Sanity check
	IF( NOT __ISVALIDREF(ConfigPDs) OR TuDestination = E_FunctionNumber.F_BEGIN_FUNCTION) THEN
		RETURN; 
	END_IF 	

	
	FOR i:=1 TO GVL_MPD.MAXPDs BY 1 DO
		//AdjacentFunctionNumbers[i] := Config_Shuttle.ConvCFG[i].eFunctionNumber;
		FOR j:=1 TO GVL_MPD.MAXDEST DO
			IF(ConfigPDs[i].PossibleDestinations[j] = TuDestination AND 
				ConfigPDs[i].eFunctionNumber <> PickupFunctionNumber (*Not possible to transfer TU to the same function*)) THEN
				M_GetDepositFunction :=ConfigPDs[i].eFunctionNumber;
				MPD_ConfigIndex:=i;
				RETURN;
			END_IF	
			IF(ConfigPDs[i].PossibleDestinations[j] = E_FunctionNumber.F_BEGIN_FUNCTION) THEN
				EXIT; //just to not iterate through alll functions to F_BEGIN_EXTERN_FUNCTION
			END_IF
		END_FOR 
	END_FOR
END_METHOD

END_FUNCTION_BLOCK

// ---- 20_Product/20_ProBox/30_Toolbox/70_Strategies/FB_MergingFiFo.TcPOU
FUNCTION_BLOCK FB_MergingFiFo
//FB_MergingFiFo 
//
VAR_INPUT
	FunctionNumber  : E_FunctionNumber;
	Disable			: BOOL; 	// Make this E_Function disabled, ie PriorityControl will not return this E_FunctionNumber
	CompareNextFunc	: E_FunctionNumber; // Check if next is set to this function. F_BEGIN_FUNCTION = No check performed		  
END_VAR

VAR_OUTPUT
	ePrevFunctionNumber		: E_FunctionNumber;		//the function number that has the highest priority to enter into Loop or intersection.	  
END_VAR
VAR CONSTANT 
    ELEMENTLAST 	: INT:=20;
	ELEMENTFIRST	: INT:=1;
	STARTZONE		: INT:=1;
	EmptyBuffer		: ST_FifoBuffer:= (eFunctionNumber:=0,EntryOK:=0, Occupied:=0) ; 
END_VAR 
VAR	
	_Buffer					: ARRAY[ELEMENTFIRST..ELEMENTLAST] OF ST_FifoBuffer;	
END_VAR
VAR_TEMP
	i						: INT;
END_VAR


ePrevFunctionNumber :=E_FunctionNumber.F_BEGIN_FUNCTION;

_M_AddItem(FunctionNumber,Disable);

//return the first item in the list (that are not disabled)
//Check if function is occupied, iterate entire buffer array
FOR i:=ELEMENTFIRST TO ELEMENTLAST BY 1 DO
	IF(_Buffer[i].EntryOK AND _Buffer[i].Occupied) THEN
		ePrevFunctionNumber :=_Buffer[i].eFunctionNumber;						
		EXIT;
	END_IF
END_FOR

METHOD PRIVATE _M_AddItem : BOOL  //FIFO table
VAR_INPUT
	FunctionNumber  : E_FunctionNumber;
	Disable			: BOOL; 	// Make this E_Function disabled, ie PriorityControl will not return this E_FunctionNumber		
END_VAR

VAR	
	myBufferIx		: INT:=0;		
	i:INT;
	j:INT;
	
END_VAR

//search for function in buffer, get myBufferIx
FOR myBufferIx := ELEMENTFIRST TO ELEMENTLAST BY 1 DO
	IF(_Buffer[myBufferIx].eFunctionNumber=FunctionNumber) THEN EXIT; END_IF
END_FOR

//if entry was not already in buffer -> search for first empty slot
IF(myBufferIx>ELEMENTLAST) THEN // no item found	
	FOR myBufferIx := ELEMENTFIRST TO ELEMENTLAST BY 1 DO
		IF(_Buffer[myBufferIx].eFunctionNumber=0) THEN EXIT;	END_IF
	END_FOR
END_IF

//if no emtpy slot was found, then buffer full, so return.
IF(myBufferIx>ELEMENTLAST) THEN RETURN; END_IF

//------------------------------------------------------------------------
// By now, the Buffer Ix is determined
// Add function number to the buffer list
//------------------------------------------------------------------------
_Buffer[myBufferIx].eFunctionNumber := FunctionNumber;
_Buffer[myBufferIx].EntryOK := NOT Disable AND _M_EntryOk(FunctionNumber);

//------------------------------------------------------------------------
// Check all functions in the list being occupied
// Check if functions being occupied
//------------------------------------------------------------------------

IF(_Buffer[myBufferIx].eFunctionNumber>0) THEN
	_Buffer[myBufferIx].Occupied:=FALSE;		
	_Buffer[myBufferIx].Occupied:=_M_Enabled(_Buffer[myBufferIx].eFunctionNumber); //check occupied and handover enabled.
	IF( NOT _Buffer[myBufferIx].Occupied) THEN
		//Clear buffer
		_Buffer[myBufferIx]:=EmptyBuffer;			
	END_IF
END_IF

//------------------------------------------------------------------------
// Sort items, 
//------------------------------------------------------------------------

_M_SortFifo();
	
_M_AddItem := TRUE;
END_METHOD

METHOD PRIVATE _M_Enabled : BOOL
VAR_INPUT
	FunctionNumber : E_FunctionNumber; 
END_VAR
VAR
	rZoneData		:REFERENCE TO ST_ZoneData;
	rZoneTrspEnable :REFERENCE TO ST_TransportEnable;	
	i:INT;
	Tu_index :DINT;
END_VAR


IF( NOT __ISVALIDREF(FunctionRegistry[FunctionNumber].rFunction)) THEN RETURN; END_IF
IF( NOT __ISVALIDREF(FunctionRegistry[FunctionNumber].rFunctionInterface)) THEN RETURN; END_IF

FOR i:=STARTZONE TO NUMBER_OF_ZONES_PER_FUNCTION BY 1 DO
	rZoneData REF= FunctionRegistry[FunctionNumber].rFunction.ZoneData[i];
	rZoneTrspEnable REF=FunctionRegistry[FunctionNumber].rFunction.ZoneInterface[i].In.Enable;	

	_M_Enabled:= _M_Enabled OR	F_PB_GetTransportControlDataRef(FunctionNumber,i).Occupied OR F_PB_GetTransportControlDataRef(FunctionNumber,i).DataPresent;
	
	IF NOT (rZoneData.AddOn.Orders.Enable AND rZoneData.AddOn.Orders.EnableHandover AND rZoneTrspEnable.HandOver AND rZoneTrspEnable.Transport) THEN
		_M_Enabled :=FALSE;
		EXIT;
	END_IF
	
	Tu_index := F_PB_GetTransportControlDataRef(FunctionNumber,i).TU_DataIndex;
	IF(Tu_index>0) THEN
		IF(NOT TU_Table.TU_DataTable[Tu_index].DataSet.JobPresent) THEN
			_M_Enabled :=FALSE;
			EXIT;
		END_IF
	END_IF
			
	//check if handover was completed, then remove from buffer
	IF(F_PB_GetTransportControlDataRef(FunctionNumber,i).eHandOverState= E_HandOverState.COMPLETE) THEN
		_M_Enabled :=FALSE;
		EXIT;
	END_IF
		
	
END_FOR
END_METHOD

METHOD PRIVATE _M_EntryOk : BOOL
VAR_INPUT
	FunctionNumber : E_FunctionNumber;	
END_VAR
VAR
	rZoneData		:REFERENCE TO ST_ZoneData;
	rZoneTrspEnable :REFERENCE TO ST_TransportEnable;
	i:INT;
	ElementNumber	: E_ElementNumber;
END_VAR
_M_EntryOk :=FALSE;
IF( NOT __ISVALIDREF(FunctionRegistry[FunctionNumber].rFunction)) THEN RETURN; END_IF
IF( NOT __ISVALIDREF(FunctionRegistry[FunctionNumber].rFunctionInterface)) THEN RETURN; END_IF
IF( NOT __ISVALIDREF(FunctionRegistry[FunctionNumber].rFunctionData)) THEN RETURN; END_IF
IF( NOT __ISVALIDREF(FunctionRegistry[FunctionNumber].rSettingsFunction)) THEN RETURN; END_IF

//check that there are no active errors in element, functon or zones

ElementNumber := FunctionRegistry[FunctionNumber].rSettingsFunction.eElementLink;
IF(__ISVALIDREF(ElementRegistry[ElementNumber].rElementData))THEN
	IF( NOT ElementRegistry[ElementNumber].rElementData.ErrorData.FunctionErrorPending AND 
		ElementRegistry[ElementNumber].rElementData.ErrorData.ErrorState <> E_ErrorState.ERROR) THEN
		_M_EntryOk :=TRUE;
	END_IF	
END_IF	



// check if element/function is started
_M_EntryOk := _M_EntryOk AND FunctionRegistry[FunctionNumber].rFunctionInterface.In.Element.OperationState.eState = E_PositionState.STARTED;								
//check if any zone/Function/element is disabled
_M_EntryOk := _M_EntryOk AND F_CheckAllEnabled(FunctionNumber);

//check that input function also has next defined (Should point to DTU but is not checked!!)
IF(THIS^.CompareNextFunc>E_FunctionNumber.F_BEGIN_FUNCTION AND FunctionRegistry[FunctionNumber].rFunctionInterface.In.eNextFunctionNumber<>CompareNextFunc) THEN
	_M_EntryOk := FALSE;
END_IF
END_METHOD

METHOD PRIVATE _M_SortFiFo : BOOL
VAR_INPUT
END_VAR
VAR
	i,j:INT;
END_VAR
FOR i:=ELEMENTFIRST TO ELEMENTLAST-1 BY 1 DO	
	IF(_Buffer[i].eFunctionNumber=0) THEN
		FOR j:=i+1 TO ELEMENTLAST BY 1 DO
			IF(_Buffer[j].eFunctionNumber <> 0) THEN
				_Buffer[i] := _Buffer[j];
				_Buffer[j] := EmptyBuffer;				
				EXIT;
			END_IF
		END_FOR
		EXIT;	//No need iterate over entire buffer. this will be covered next cycle.
	END_IF	
END_FOR
END_METHOD

METHOD PUBLIC M_GetFifoIndex : E_FunctionNumber
VAR_INPUT
	Index:INT; // 1 is the most prioritized Function
END_VAR
VAR
	myIndex,ix,i:INT;	
END_VAR

IF(Index<ELEMENTFIRST) THEN
	myIndex:= ELEMENTFIRST;
ELSIF(Index>ELEMENTLAST) THEN
	myIndex:= ELEMENTLAST;
ELSE
	myIndex:=Index;
END_IF


//return the first item in the list (that are not disabled)
//Check if function is occupied, iterate all zones
FOR i:=ELEMENTFIRST TO ELEMENTLAST BY 1 DO
	IF(_Buffer[i].EntryOK AND _Buffer[i].Occupied) THEN
		ix:= ix+1;
		IF(ix=myIndex) THEN
			M_GetFifoIndex :=_Buffer[i].eFunctionNumber;
			EXIT;
		END_IF			
	END_IF
END_FOR
END_METHOD

//Set function to the lowest priority, ie move to last positoin in FIFO
METHOD PUBLIC M_MoveToLast : BOOL
VAR_INPUT
	FunctionNumber : E_FunctionNumber;
	//Index:INT;	
END_VAR
VAR
	i:INT;
	MyIndex:Int;
END_VAR
IF(FunctionNumber=0) THEN RETURN; END_IF

//return the first item in the list (that are not disabled)
//Check if function is occupied, iterate all zones
FOR i:=ELEMENTFIRST TO ELEMENTLAST BY 1 DO
	IF(_Buffer[i].eFunctionNumber = FunctionNumber) THEN
		//Clear buffer -> remove from FIFO-> it will be added next cycle
		_Buffer[i]:=EmptyBuffer;
		EXIT;				
	END_IF
END_FOR

//sort fifo (_M_SortFiFo()) not needed, this will be carried out when re-adding the unit
END_METHOD

END_FUNCTION_BLOCK

// ---- 20_Product/20_ProBox/30_Toolbox/F_CheckAllEnabled.TcPOU
FUNCTION F_CheckAllEnabled : BOOL
(**************************************************************************************
 * 	Application		:	BoxControl Framework
 *	Revision		:	$Revision: 417092 $
 *	Revision date	:	$Date: 2018-11-14 12:58:58 +0100 (Mi., 14 Nov 2018) $
 *	Last changed by	:	$Author: q8aberh $
 *	URL				:	$URL: http://almscdc.swisslog.com/repo/SWPD/Development/ProMove/02_Controls/ProBox/03_Implementation/01_DevelopmentProject/01_Software/ProBox_COE/ProBox_DevProj_v1.0/PLC_1/20_Product/10_App/12_E_Functions/11_ProBox/02_Functions/02_TransportControl/F_Che $
 *
 *	Purpose			:	Returns true if all the zones on the function are enabled
 *
 * ------------------------------------------------------------------------------------
 *	Copyright Swisslog [IP AG], Switzerland. All rights reserved.
 * 
 * ------------------------------------------------------------------------------------
 *	
 * 	Revision History: 
 *
 * 	VERSION			DATE			INITIALS			DESCRIPTION
 *	0.1				2018-09-17		PkF					First version
 *
 **************************************************************************************)
VAR_INPUT
	eFunctionNumber		: E_FunctionNumber; // Function number
END_VAR
VAR
	idx 				: INT; // Iterator
	AllEnabled			: BOOL; // Temp to check if all zones are enabled
	ElementNumber		: E_ElementNumber;
END_VAR

// Check if function number is valid
IF eFunctionNumber > E_FunctionNumber.F_BEGIN_FUNCTION AND
   eFunctionNumber < E_FunctionNumber.F_END_FUNCTION THEN
  
	// Check reference is valid
	IF  __ISVALIDREF(FunctionRegistry[eFunctionNumber].rSettingsFunction) AND 
		__ISVALIDREF(FunctionRegistry[eFunctionNumber].rFunctionData) THEN
		// Return All Started
		AllEnabled := TRUE;
		FOR idx := 1 TO FunctionRegistry[eFunctionNumber].rSettingsFunction.NumberOfZones DO
			IF NOT Functionregistry[eFunctionNumber].Zone[idx].refZoneInterface.In.ZoneEnable  THEN
				AllEnabled := FALSE;
				EXIT;
			END_IF
		END_FOR
		F_CheckAllEnabled := AllEnabled;
								
		//check if function or element is disabled.				
		IF(__ISVALIDREF(FunctionRegistry[eFunctionNumber].rFunctionInterface)) THEN
			F_CheckAllEnabled := F_CheckAllEnabled AND FunctionRegistry[eFunctionNumber].rFunctionInterface.In.FunctionEnable;
		END_IF
		ElementNumber := FunctionRegistry[eFunctionNumber].rSettingsFunction.eElementLink;
		IF(__ISVALIDREF(ElementRegistry[ElementNumber].rElementInterface)) THEN
			F_CheckAllEnabled := F_CheckAllEnabled AND ElementRegistry[ElementNumber].rElementInterface.In.ElementEnable;	
		END_IF
	END_IF
   
	
	  
     
   
END_IF

END_FUNCTION

// ---- 20_Product/20_ProBox/30_Toolbox/F_PB_GetAdjacentFunctionZoneIndex.TcPOU
//Get the Zone index of a adjecent function.
//Return: TRUE if conditions are met and ZoneIndex is valid. FALSE: conditions not met. 
FUNCTION F_PB_GetAdjacentFunctionZoneIndex : BOOL
VAR_INPUT
	CheckFunction			: E_FunctionNumber; // The adjacent function number
	ExpectedFunction		: E_FunctionNumber;	// The function that the adjecent function shall be compared with		
	RequireNextDefined		:BOOL;				// Require that the CheckFunction has defined next towards the CheckFunction function
	RequirePreviousDefined	:BOOL;				// Require that the CheckFunction function has defined previous towards the CheckFunction function
END_VAR
VAR_IN_OUT
	ZoneIndex	: INT;	
END_VAR
VAR
END_VAR

	F_PB_GetAdjacentFunctionZoneIndex:=FALSE;
	ZoneIndex:=0;
		
	//Sanity check
	IF(ExpectedFunction =0) THEN RETURN; END_IF
	IF(CheckFunction =0) THEN RETURN; END_IF
	IF(NOT __ISVALIDREF(FunctionRegistry[CheckFunction].rSettingsFunction)) THEN RETURN; END_IF
	IF(NOT __ISVALIDREF(FunctionRegistry[CheckFunction].rFunctionInterface)) THEN RETURN; END_IF
	IF(NOT __ISVALIDREF(FunctionRegistry[ExpectedFunction].rFunctionInterface)) THEN RETURN; END_IF
	
	//check that F_Handover has defined F_Takever as its next function
	IF(RequireNextDefined AND FunctionRegistry[CheckFunction].rFunctionInterface.In.eNextFunctionNumber <> ExpectedFunction) THEN
		RETURN; //the handover function has not set next towards the takeover function.
	END_IF
	//Check that F_Takeover has define F_Handover as its previous function
	IF(RequirePreviousDefined AND FunctionRegistry[CheckFunction].rFunctionInterface.In.ePrevFunctionNumber <> ExpectedFunction) THEN
		RETURN; //the handover function has not set next towards the takeover function.
	END_IF			

	IF( FunctionRegistry[CheckFunction].rSettingsFunction.eAdjacentFunctionNumberSide[1] = ExpectedFunction OR
		FunctionRegistry[CheckFunction].rSettingsFunction.eAdjacentFunctionNumberSide[3] = ExpectedFunction) THEN
		ZoneIndex := 1;
		F_PB_GetAdjacentFunctionZoneIndex:=TRUE;
		
	ELSIF(FunctionRegistry[CheckFunction].rSettingsFunction.eAdjacentFunctionNumberSide[2] = ExpectedFunction OR
		  FunctionRegistry[CheckFunction].rSettingsFunction.eAdjacentFunctionNumberSide[4] = ExpectedFunction) THEN
		
		IF(FunctionRegistry[CheckFunction].rSettingsFunction.NumberOfZones<= Conveyor.NUMBER_OF_ZONES_PER_FUNCTION) THEN
			ZoneIndex := FunctionRegistry[CheckFunction].rSettingsFunction.NumberOfZones;
			F_PB_GetAdjacentFunctionZoneIndex:=TRUE;
		END_IF
	END_IF

END_FUNCTION

// ---- 20_Product/20_ProBox/22_ProMove/03_Controls/13_ExtendedRunControl/FB_ExtendedRun.TcPOU
//Extended run means that an TU can run beyond the stop sensor until the TU raches the extended run stop sensor
//The conveyor starts when next function is determined.
FUNCTION_BLOCK PUBLIC FB_ExtendedRun
VAR_INPUT
	HostFunction	: E_FunctionNumber;	//Function  number of the element that shall run extended run	
	HWSensorStop	: BOOL; //the actual HW sensor input that shall stop the extended run
	Enable			: BOOL; //The extended run will start when Enable signal is true, possible to delay the start of the transfer towards ExtRunStop sensor
	Config			: REFERENCE TO ST_CFG_ExtendedRun;
END_VAR
VAR_OUTPUT
	ExtRunStarted:BOOL;	//TRUE = Extended run functionality started->For functions to disable TransportEnableHandOver	
	ExtRunSynteticSensor:BOOL;	//Signal representing an TU Occupied sensor.
END_VAR
VAR_IN_OUT
	ErrorData 				: ST_ErrorDataSet; // Error data
	//FunctionOrders			: ST_FunctionOrders;
END_VAR
VAR	
	_StartTrig:R_TRIG;	
	_DriveTimeout : TON;
	_State:INT;
	_ExtRunDrive:BOOL;
	_ExtRunError:BOOL;
	
	//property
	_pOverrideNextUnDef	: BOOL := FALSE; //TRUE:= Next is not required to start extended run, not recomended for DTU.
END_VAR
VAR_TEMP
	Occupied:BOOL;
	EnableDrive:BOOL;		
	TakeingOver:BOOL;
	
END_VAR
VAR CONSTANT 
	EXTRUN_IDLE:INT :=1; //Idleing...
	EXTRUN_WAIT:INT :=2; //Wait for enable signal
	EXTRUN_BUSY:INT :=3; //Busy driving element
	EXTRUN_DONE:INT :=0; //Complete
END_VAR


//SanityCheck
IF( NOT __ISVALIDREF(FunctionRegistry[HostFunction].rFunctionData) OR 
	NOT __ISVALIDREF(FunctionRegistry[HostFunction].rFunctionInterface) OR
	Config.FunctionZone<=0 OR NOT Config.Activated) THEN
	ExtRunStarted:=ExtRunSynteticSensor:=FALSE;
	RETURN;
END_IF


Occupied := F_PB_GetTransportControlDataRef(HostFunction,Config.FunctionZone).Occupied;
TakeingOver := _M_CheckConditionsPreCheckState();

CASE _State OF
	EXTRUN_IDLE:			
		IF(_M_CheckConditionsBusyState(Occupied,NOT TakeingOver AND ErrorData.ErrorType <> E_ErrorType.ERROR)) THEN
			_State:=EXTRUN_WAIT; //Wait for Enable signal, but set Busy, in order to disable handover for the function		 
		END_IF
	EXTRUN_WAIT:
		IF(NOT Occupied OR Enable) THEN
			_State:=EXTRUN_BUSY; //Start element driving
		END_IF
	EXTRUN_BUSY:
		IF(NOT Occupied OR HWSensorStop) THEN
			_State:=EXTRUN_DONE; //extended run complete
		END_IF
	EXTRUN_DONE: 
		IF(NOT Occupied) THEN
			_State:=EXTRUN_IDLE; //Idle
		END_IF			
END_CASE


// ---------------------------------------------------
//Set output
// ---------------------------------------------------
ExtRunStarted := _State=EXTRUN_BUSY OR _State=EXTRUN_WAIT OR TakeingOver; //For functions to disable TransportEnableHandOver;
ExtRunSynteticSensor := (HWSensorStop OR _State=EXTRUN_BUSY) AND NOT TakeingOver;//Disabled during takeover, sine we dont want the transfer to stop if ext.run sensor is blocked


// ---------------------------------------------------
// Set errors
// ---------------------------------------------------
F_ResetError(FALSE,ErrorData);
//Check Timeout
_DriveTimeout(IN:= _ExtRunDrive, PT:=Config.TimeoutDriveRun);
IF(_DriveTimeout.Q) THEN	
	F_SetError(E_ErrorType.ERROR,'Timeout reaching extended run stop sensor',E_ErrorConv.TIMEOUT_MOVEMENT, ErrorData);
END_IF

//check if stopsensor is blocked when starting an extended run
_StartTrig(CLK:=_State=EXTRUN_BUSY AND _ExtRunDrive);
IF(_StartTrig.Q  AND HWSensorStop) THEN
	F_SetError(E_ErrorType.ERROR,'Extended run stop sensor blocked',E_ErrorConv.POSITION_OCCUPIED_BEFORE_TAKEOVER, ErrorData);	
	_State:=EXTRUN_IDLE; //start over
END_IF


_ExtRunError := ErrorData.ErrorType = E_ErrorType.ERROR;

METHOD PRIVATE _M_CheckConditionsBusyState : BOOL
VAR_INPUT
	Occupied:BOOL;
	Enabled:BOOL;
END_VAR
//Start conditions

IF( NOT Enabled OR NOT Occupied OR NOT Config.Activated OR
	FunctionRegistry[HostFunction].rFunctionData.OperationState.eMode <> E_PositionMode.AUTO_MODE OR
	FunctionRegistry[HostFunction].rFunctionData.ErrorData.ErrorState = E_ErrorState.ERROR OR
	FunctionRegistry[HostFunction].rFunctionData.ErrorData.ZoneErrorPending OR	
	FunctionRegistry[HostFunction].rFunctionData.OperationState.eState <> E_PositionState.STARTED) THEN
	RETURN;
END_IF

IF(_pOverrideNextUnDef) THEN
	_M_CheckConditionsBusyState :=TRUE;

//check that nextfunction is determined
ELSIF(FunctionRegistry[HostFunction].rFunctionInterface.In.eNextFunctionNumber<> E_FunctionNumber.F_BEGIN_FUNCTION) THEN
	//determine if next function is on the sided configured with RunAxis config parameter
	CASE Config.ElementRunAxis OF
		E_Axis_Orientation.Element_12:
			_M_CheckConditionsBusyState:= FunctionRegistry[HostFunction].rFunctionInterface.In.eNextFunctionNumber = FunctionRegistry[HostFunction].rSettingsFunction.eAdjacentFunctionNumberSide[2];			 
		E_Axis_Orientation.Element_21:
			_M_CheckConditionsBusyState:= FunctionRegistry[HostFunction].rFunctionInterface.In.eNextFunctionNumber = FunctionRegistry[HostFunction].rSettingsFunction.eAdjacentFunctionNumberSide[1];			
		E_Axis_Orientation.Element_34:
			_M_CheckConditionsBusyState:= FunctionRegistry[HostFunction].rFunctionInterface.In.eNextFunctionNumber = FunctionRegistry[HostFunction].rSettingsFunction.eAdjacentFunctionNumberSide[4];			
		E_Axis_Orientation.Element_43:
			_M_CheckConditionsBusyState:= FunctionRegistry[HostFunction].rFunctionInterface.In.eNextFunctionNumber = FunctionRegistry[HostFunction].rSettingsFunction.eAdjacentFunctionNumberSide[3];				
	END_CASE
END_IF
END_METHOD

METHOD PRIVATE _M_CheckConditionsPreCheckState : BOOL
VAR_INPUT
END_VAR
VAR
END_VAR
//check if takeover is active, (ignored when simultaneous mode is active)
_M_CheckConditionsPreCheckState :=  (F_PB_GetTransportControlDataRef(HostFunction,Config.FunctionZone).eTakeOverState = E_TakeOverState.ACTIVE OR
									 F_PB_GetTransportControlDataRef(HostFunction,Config.FunctionZone).eTakeOverState = E_TakeOverState.COMPLETE) AND
									 (F_PB_GetTransportControlDataRef(HostFunction,Config.FunctionZone).eTransportState <> E_TransportState.SIMULTANEOUS AND
									  F_PB_GetTransportControlDataRef(HostFunction,Config.FunctionZone).eTransportState <> E_TransportState.SIMULTANEOUS_OCCUPIED);
END_METHOD

//Set enable status on correct axis
METHOD PRIVATE _M_FunctionOrder : BOOL
VAR_INPUT	
	ExtRunError:BOOL; //True = extended run function has error
	Enabled:BOOL; //Conditions ok for driving motor
END_VAR
VAR_IN_OUT
	FunctionOrders			: ST_FunctionOrders;
END_VAR


// Check that input functionorder is enable drive, ie do not override host function

//determine if next function is on the sided configured with RunAxis config parameter
CASE Config.ElementRunAxis OF
	E_Axis_Orientation.Element_12, E_Axis_Orientation.Element_21:			
		FunctionOrders.Enable := FunctionOrders.Enable AND Enabled AND NOT ExtRunError;
		_M_FunctionOrder := FunctionOrders.Enable;				 
	
	E_Axis_Orientation.Element_34, E_Axis_Orientation.Element_43:			
		FunctionOrders.Enable_34 := FunctionOrders.Enable_34 AND Enabled AND NOT ExtRunError;
		_M_FunctionOrder := FunctionOrders.Enable_34;
		
END_CASE
END_METHOD

//Set enable status on correct axis
METHOD PUBLIC M_SetProBoxFunctionOrder : BOOL
VAR_IN_OUT
	FunctionOrders			: ST_FunctionOrders;
END_VAR
VAR
	EnableDrive:BOOL;
	ErrorActive:BOOL;
END_VAR

_ExtRunDrive:=FALSE;
ErrorActive :=FALSE;
IF(__ISVALIDREF(FunctionRegistry[HostFunction].rFunctionData)) THEN
	ErrorActive := FunctionRegistry[HostFunction].rFunctionData.ErrorData.ErrorState = E_ErrorState.ERROR OR _ExtRunError;
END_IF

//Get host function enable drive signals, and apply own enable signals
IF(_State=EXTRUN_BUSY) THEN
	EnableDrive := _M_FunctionOrder(ErrorActive,Enable, FunctionOrders :=FunctionOrders);

	_ExtRunDrive := EnableDrive AND		 
			 FunctionRegistry[HostFunction].rFunctionData.OperationState.eMode = E_PositionMode.AUTO_MODE AND
			 FunctionRegistry[HostFunction].rFunctionData.ErrorData.ErrorState <> E_ErrorState.ERROR AND 
			(FunctionRegistry[HostFunction].rFunctionData.OperationState.eState =E_PositionState.STARTED OR
			 FunctionRegistry[HostFunction].rFunctionData.OperationState.eState =E_PositionState.STOPPING); 
		 
END_IF

IF(_ExtRunDrive) THEN
    FunctionOrders := F_ProBoxToFunctionOrders(
                        CreepSpeed_12	:= Config.DriveSpeed = E_ProBoxMotorSpeed.CREEP_SPEED, 
                        LowSpeed_12 	:= Config.DriveSpeed = E_ProBoxMotorSpeed.LOW_SPEED,
                        CreepSpeed_34 	:= Config.DriveSpeed = E_ProBoxMotorSpeed.CREEP_SPEED, 
                        LowSpeed_34 	:= Config.DriveSpeed = E_ProBoxMotorSpeed.LOW_SPEED, 
                        Forward_12		:= _ExtRunDrive AND Config.ElementRunAxis = E_Axis_Orientation.Element_12, 
                        Reverse_12 		:= _ExtRunDrive AND Config.ElementRunAxis = E_Axis_Orientation.Element_21,	
                        Forward_34 		:= _ExtRunDrive AND Config.ElementRunAxis = E_Axis_Orientation.Element_34, 
                        Reverse_34 		:= _ExtRunDrive AND Config.ElementRunAxis = E_Axis_Orientation.Element_43,
                        Enable_12		:= FunctionOrders.Enable,
                        Enable_34		:= FunctionOrders.Enable_34);
END_IF
END_METHOD

//Enable extended run without having next function defined
//TRUE:= Next is not required to be defined in order to start extended run.
//Not recomended for DTU's
PROPERTY PUBLIC P_OverrideNextUnDef : BOOL
SET
_pOverrideNextUnDef	:= P_OverrideNextUnDef;
END_SET
END_PROPERTY

END_FUNCTION_BLOCK

// ---- 20_Product/20_ProBox/22_ProMove/03_Controls/F_ProBoxToFunctionOrders.TcPOU
FUNCTION F_ProBoxToFunctionOrders : ST_FunctionOrders
VAR_INPUT
	CreepSpeed_12 	: BOOL;	
	LowSpeed_12 	: BOOL;
	Forward_12 		: BOOL;	
	Reverse_12 		: BOOL;	
	CreepSpeed_34 	: BOOL;	
	LowSpeed_34 	: BOOL;
	Forward_34 		: BOOL;	
	Reverse_34 		: BOOL;	
	Enable_12		: BOOL;
	Enable_34		: BOOL;
END_VAR

// Convert ProBox motor speeds to "BCF" speeds just to avoid chainging the interfaces between functions and elements.
IF CreepSpeed_12 THEN
	F_ProBoxToFunctionOrders.ReqSpeed := 20;
ELSIF LowSpeed_12 THEN
	F_ProBoxToFunctionOrders.ReqSpeed := 50;
ELSE
	F_ProBoxToFunctionOrders.ReqSpeed := 100;
END_IF;

IF CreepSpeed_34 THEN
	F_ProBoxToFunctionOrders.ReqSpeed_34 := 20;
ELSIF LowSpeed_34 THEN
	F_ProBoxToFunctionOrders.ReqSpeed_34 := 50;
ELSE
	F_ProBoxToFunctionOrders.ReqSpeed_34 := 100;
END_IF;

IF Forward_12 THEN
	F_ProBoxToFunctionOrders.ReqDriveDirection := TRUE;
//ELSIF Reverse_12 THEN
ELSE
	F_ProBoxToFunctionOrders.ReqDriveDirection := FALSE;
END_IF;

IF Forward_34 THEN
	F_ProBoxToFunctionOrders.ReqDriveDirection_34 := TRUE;
//ELSIF Reverse_34 THEN
ELSE
	F_ProBoxToFunctionOrders.ReqDriveDirection_34 := FALSE;
END_IF;

F_ProBoxToFunctionOrders.ReqDriveRun := Forward_12 OR Reverse_12;
F_ProBoxToFunctionOrders.ReqDriveRun_34 := Forward_34 OR Reverse_34;
F_ProBoxToFunctionOrders.Enable := Enable_12;
F_ProBoxToFunctionOrders.Enable_34 := Enable_34;

END_FUNCTION

// ---- 20_Product/20_ProBox/22_ProMove/03_Controls/FB_ProBoxToElementState.TcPOU
FUNCTION_BLOCK FB_ProBoxToElementState
VAR_INPUT
	CreepSpeed_12 	: BOOL;	
	LowSpeed_12 	: BOOL;
	Forward_12 		: BOOL;	
	Reverse_12 		: BOOL;	
	CreepSpeed_34 	: BOOL;	
	LowSpeed_34 	: BOOL;
	Forward_34 		: BOOL;	
	Reverse_34 		: BOOL;
END_VAR

VAR_OUTPUT
	ElementState : ST_ElementState;
END_VAR


// Convert ProBox motor speeds to "BCF" speeds just to avoid chainging the interfaces between functions and elements.
IF CreepSpeed_12 THEN
	ElementState.Speed := 20;
ELSIF LowSpeed_12 THEN
	ElementState.Speed := 50;
ELSE
	ElementState.Speed := 100;
END_IF;

IF CreepSpeed_34 THEN
	ElementState.Speed_34 := 20;
ELSIF LowSpeed_34 THEN
	ElementState.Speed_34 := 50;
ELSE
	ElementState.Speed_34 := 100;
END_IF;
	

IF Forward_12 THEN
	ElementState.DriveDirection := TRUE;
ELSIF Reverse_12 THEN
	ElementState.DriveDirection := FALSE;
END_IF;

IF Forward_34 THEN
	ElementState.DriveDirection_34 := TRUE;
ELSIF Reverse_34 THEN
	ElementState.DriveDirection_34 := FALSE;
END_IF;


ElementState.DriveRunning := Forward_12 OR Reverse_12;
ElementState.DriveRunning_34 := Forward_34 OR Reverse_34;

END_FUNCTION_BLOCK

// ---- 20_Product/20_ProBox/22_ProMove/11_Addons/FB_AddOnErrHandler.TcPOU
FUNCTION_BLOCK INTERNAL FB_AddOnErrHandler
VAR_INPUT
	AddOnSettingsFunction 	: REFERENCE TO ST_CFG_Function;
	AddOnFunctionData		: REFERENCE TO ST_FunctionData;
END_VAR
VAR_OUTPUT
END_VAR
VAR
	//_ParentZoneErrorData        :ST_ZoneErrorStruct;
	_ParentZoneErrorActive      : BOOL;								//Last cycle error state of the main function
	LinkedZoneErrorStruct	: REFERENCE TO ST_ZoneErrorStruct;	//zone error of the main function that owns the AddOn
	i 							: INT;
	LinkedFuncNumber 			: E_FunctionNumber;					//Function number of the functino that owns the AddOn	
	LinkedZoneNumber 			: INT;								//Zone number that the AddOn is linked to
	
END_VAR

(**************************************************************************************
 * 	NAME		FB_AddOnErrHandler
 * 	FUNCTION	Should only be called from AddOns after the call to the A_ErrorHandler();
 				This function adds the AddOn functionData error to the function that the
				AddOn is linked to and reset the error if it was acknowledged from 
				Sync visualization or reset button.
				Note, if the AddOn can be acknowleded by Sync (ie Scanner) then this 
				functionblock should not be called.				
 **************************************************************************************)

// Part 1
// -Check if parent function that owns the add-on is going from "error"  to "no error pending"
//  -if so, then it was probably acknowledged by operator via sync or manual button on switching group
	
	// Sanity checks	
	IF(NOT __ISVALIDREF(AddOnSettingsFunction) OR NOT __ISVALIDREF(AddOnFunctionData) ) THEN
		RETURN;
	END_IF

	LinkedFuncNumber 	:= AddOnSettingsFunction.FunctionLink.eFunctionNumber;
	LinkedZoneNumber	:= AddOnSettingsFunction.FunctionLink.ZoneNumber;
		
	// Check zoneNumber is within valid range
	IF(LinkedZoneNumber=0 OR LinkedZoneNumber>NUMBER_OF_ZONES_PER_FUNCTION) THEN
		F_SetExternalElementError(AddOnSettingsFunction.eElementLink,E_ErrorType.ERROR,'Check Function link on Addons', E_ErrorConv.CONFIGURATION_ERROR);
		RETURN;
	END_IF
	//check reference is valid
	IF(NOT __ISVALIDREF(FunctionRegistry[LinkedFuncNumber].rFunctionData) ) THEN
		RETURN;
	END_IF	
	//Check reference is valid
	IF(NOT __ISVALIDREF(FunctionRegistry[LinkedFuncNumber].Zone[LinkedZoneNumber].refZoneData) ) THEN
		RETURN;
	END_IF
	LinkedZoneErrorStruct REF= FunctionRegistry[LinkedFuncNumber].Zone[LinkedZoneNumber].refZoneData.ErrorData; 
		
	IF(_ParentZoneErrorActive AND LinkedZoneErrorStruct.Error.ErrorType = E_ErrorType.NO_ERROR_PENDING) THEN
		FOR i:=1 TO NUMBER_OF_ERROR_SETS DO
			AddOnFunctionData.ErrorData.ErrorDataSet[i].ResetError:=TRUE;
		END_FOR
		//Reset external errors on the function that the AddOn is linked to
		F_ResetExternalFunctionError(	eFunctionNumber := LinkedFuncNumber, ZoneNumber := LinkedZoneNumber, Reset := FALSE);	
                
// Part 2.
//  -Add the AddOn error to the function zone that owns the Addon
	ELSIF(AddOnFunctionData.ErrorData.Error.ErrorType = E_ErrorType.ERROR AND LinkedZoneErrorStruct.Error.ErrorType = E_ErrorType.NO_ERROR_PENDING) THEN
		F_SetExternalFunctionError(
								   eFunctionNumber := AddOnSettingsFunction.FunctionLink.eFunctionNumber,
								   ZoneNumber := 	AddOnSettingsFunction.FunctionLink.ZoneNumber,
								   ErrorType            := AddOnFunctionData.ErrorData.Error.ErrorType,								  
								   ErrorParam	:= CONCAT(CONCAT(AddOnSettingsFunction.FunctionName,': '),AddOnFunctionData.ErrorData.Error.ErrorParam),
								   ErrorMsg             := AddOnFunctionData.ErrorData.Error.ErrorCode.Conv); 
	END_IF
	
	//Get errostate of parentZone	
	_ParentZoneErrorActive := LinkedZoneErrorStruct.Error.ErrorType = E_ErrorType.ERROR;

END_FUNCTION_BLOCK

// ---- 20_Product/20_ProBox/22_ProMove/14_Groups/10_App/F_DebugUseEmuVizu.TcPOU
FUNCTION F_DebugUseEmuVizu : BOOL
VAR_IN_OUT
	SGref			: FB_ProBOXSG; //Reference to Switching group
	SG_Emuref		: FB_ProBOXSG_Emulation; //Reference to emulation switching group
END_VAR

//usage
// F_DebugUseEmuVizu(Groups.fbSG_001,GroupsEmulation.fbSG_001_Emulation)


SGref.HW_Inputs.AK.OpResetError		:= SGref.HW_Inputs.AK.OpResetError 	OR SG_Emuref.DebugResetButton;
SGref.HW_Inputs.AK.OpAutoOn			:= SGref.HW_Inputs.AK.OpAutoOn 		OR SG_Emuref.DebugStartButton;
SGref.HW_Inputs.AK.OpMcOn			:= SGref.HW_Inputs.AK.OpMcOn 		OR SG_Emuref.DebugMcOnButton;
SGref.HW_Inputs.AK.OpResetSafety	:= SGref.HW_Inputs.AK.OpResetSafety	OR SG_Emuref.DebugResetEmgButton;
SGref.HW_Inputs.AK.OpManAuto		:= SGref.HW_Inputs.AK.OpManAuto	AND NOT SG_Emuref.DebugManualModeSw;

END_FUNCTION

// ---- 20_Product/20_ProBox/30_Toolbox/11_Emu/F_AddPhysicalTU.TcPOU
FUNCTION F_AddPhysicalTU : BOOL
(**************************************************************************************
 * 	Application		:	BoxControl Framework
 *	Revision		:	$Revision:  $
 *	Revision date	:	$Date: $
 *	Last changed by	:	$Author: $
 *	URL				:	$URL: $
 *
 *	Purpose			:	Adds physical (emulation) TU data (equal to ATQ)
 *
 * ------------------------------------------------------------------------------------
 *	Copyright Swisslog [IP AG], Switzerland. All rights reserved.
 * 
 * ------------------------------------------------------------------------------------
 *	
 * 	Revision History: 
 *
 * 	VERSION			DATE			INITIALS			DESCRIPTION
 *	0.1				01.01.2001		swl					Example
 *
 **************************************************************************************)
VAR_INPUT
	eFunctionNumber : E_FunctionNumber;
	ZoneNumber		: INT;
	(*Height
	Length
	Weight
	Width *)
	
END_VAR
VAR
	mName	: STRING;
	NewID 	: T_MaxString;
END_VAR
VAR_STAT
	ID		: INT := 1;
	ATQ		: ST_ITC_ATQ;
END_VAR

mName := F_GetFunctionName(eFunctionNumber:= eFunctionNumber, ZoneNumber:= ZoneNumber);
ATQ.Position := F_ReduceToAlphaNumeric(InputString := mName);

NewID := F_StuffString(
			InputString 	:= INT_TO_STRING(ID), 
			StringLength	:= 8, 
			StuffCharacter 	:= '0',
			LeftAligned     := FALSE);
			
ID := ID + 1;

IF ID > 9998 THEN
	ID := 1;
END_IF

